LIN {X 0,Y 143.215,Z 734.624,A -85,B 0,C 180,E1 -24462.047,E2 -24462.047} C_VEL
LIN {X 0,Y 143.54,Z 734.586,A -85,B 0,C 180,E1 -24468.706,E2 -24468.706} C_VEL
LIN {X 0,Y 143.596,Z 734.591,A -85,B 0,C 180,E1 -24471.557,E2 -24471.557} C_VEL
LIN {X 0,Y 144.126,Z 734.536,A -85,B 0,C 180,E1 -24480,E2 -24480} C_VEL
LIN {X 0,Y 143.584,Z 734.584,A -85,B 0,C 180,E1 -24488.444,E2 -24488.444} C_VEL
LIN {X 0,Y 143.385,Z 734.625,A -85,B 0,C 180,E1 -24492.741,E2 -24492.741} C_VEL
LIN {X 0,Y 143.397,Z 734.844,A -85,B 0,C 180,E1 -24493.461,E2 -24493.461} C_VEL
LIN {X 0,Y 144.593,Z 738.379,A -85,B 0,C 180,E1 -24498.325,E2 -24498.325} C_VEL
LIN {X 0,Y 149.594,Z 746.195,A -85,B 0,C 180,E1 -24504.088,E2 -24504.088} C_VEL
LIN {X 0,Y 150.898,Z 748.17,A -85,B 0,C 180,E1 -24505.335,E2 -24505.335} C_VEL
LIN {X 0,Y 155.689,Z 755.868,A -85,B 0,C 180,E1 -24509.397,E2 -24509.397} C_VEL
LIN {X 0,Y 159.728,Z 762.939,A -85,B 0,C 180,E1 -24512.355,E2 -24512.355} C_VEL
LIN {X 0,Y 163.362,Z 769.766,A -85,B 0,C 180,E1 -24514.752,E2 -24514.752} C_VEL
LIN {X 0,Y 166.388,Z 775.905,A -85,B 0,C 180,E1 -24516.604,E2 -24516.604} C_VEL
LIN {X 0,Y 170.599,Z 785.165,A -85,B 0,C 180,E1 -24519.003,E2 -24519.003} C_VEL
LIN {X 0,Y 175.203,Z 796.764,A -85,B 0,C 180,E1 -24521.461,E2 -24521.461} C_VEL
LIN {X 0,Y 175.895,Z 798.887,A -85,B 0,C 180,E1 -24521.832,E2 -24521.832} C_VEL
LIN {X 0,Y 177.097,Z 822.748,A -85,B 0,C 180,E1 -24523.616,E2 -24523.616} C_VEL
LIN {X 0,Y 177.866,Z 846.501,A -85,B 0,C 180,E1 -24525.184,E2 -24525.184} C_VEL
LIN {X 0,Y 176.539,Z 862.826,A -85,B 0,C 180,E1 -24525.881,E2 -24525.881} C_VEL
LIN {X 0,Y 174.42,Z 875.839,A -85,B 0,C 180,E1 -24526.79,E2 -24526.79} C_VEL
LIN {X 0,Y 171.762,Z 887.436,A -85,B 0,C 180,E1 -24527.956,E2 -24527.956} C_VEL
LIN {X 0,Y 168.154,Z 899.75,A -85,B 0,C 180,E1 -24529.647,E2 -24529.647} C_VEL
LIN {X 0,Y 164.16,Z 910.742,A -85,B 0,C 180,E1 -24531.651,E2 -24531.651} C_VEL
LIN {X 0,Y 160.406,Z 919.713,A -85,B 0,C 180,E1 -24533.761,E2 -24533.761} C_VEL
LIN {X 0,Y 156.192,Z 928.978,A -85,B 0,C 180,E1 -24536.574,E2 -24536.574} C_VEL
LIN {X 0,Y 151.739,Z 938.048,A -85,B 0,C 180,E1 -24540.161,E2 -24540.161} C_VEL
LIN {X 0,Y 147.966,Z 945.838,A -85,B 0,C 180,E1 -24544.259,E2 -24544.259} C_VEL
LIN {X 0,Y 144.95,Z 952.191,A -85,B 0,C 180,E1 -24548.697,E2 -24548.697} C_VEL
LIN {X 0,Y 143.145,Z 956.745,A -85,B 0,C 180,E1 -24552.888,E2 -24552.888} C_VEL
LIN {X 0,Y 142.563,Z 958.65,A -85,B 0,C 180,E1 -24555.055,E2 -24555.055} C_VEL
LIN {X 0,Y 141.552,Z 960.306,A -85,B 0,C 180,E1 -24557.308,E2 -24557.308} C_VEL
LIN {X 0,Y 138.628,Z 962.218,A -85,B 0,C 180,E1 -24561.1,E2 -24561.1} C_VEL
LIN {X 0,Y 136.461,Z 963.168,A -85,B 0,C 180,E1 -24564.281,E2 -24564.281} C_VEL
LIN {X 0,Y 135.714,Z 963.596,A -85,B 0,C 180,E1 -24566.766,E2 -24566.766} C_VEL
LIN {X 0,Y 135.734,Z 963.691,A -85,B 0,C 180,E1 -24567.604,E2 -24567.604} C_VEL
LIN {X 0,Y 136.146,Z 963.933,A -85,B 0,C 180,E1 -24570.02,E2 -24570.02} C_VEL
LIN {X 0,Y 135.66,Z 963.612,A -85,B 0,C 180,E1 -24572.989,E2 -24572.989} C_VEL
LIN {X 0,Y 135.089,Z 961.834,A -85,B 0,C 180,E1 -24578.706,E2 -24578.706} C_VEL
LIN {X 0,Y 135.494,Z 959.18,A -85,B 0,C 180,E1 -24583.517,E2 -24583.517} C_VEL
LIN {X 0,Y 136.879,Z 955.695,A -85,B 0,C 180,E1 -24587.962,E2 -24587.962} C_VEL
LIN {X 0,Y 139.288,Z 951.174,A -85,B 0,C 180,E1 -24592.255,E2 -24592.255} C_VEL
LIN {X 0,Y 140.522,Z 949.425,A -85,B 0,C 180,E1 -24593.8,E2 -24593.8} C_VEL
LIN {X 0,Y 144.564,Z 949.723,A -85,B 0,C 180,E1 -24599.107,E2 -24599.107} C_VEL
LIN {X 0,Y 150.41,Z 949.085,A -85,B 0,C 180,E1 -24604.123,E2 -24604.123} C_VEL
LIN {X 0,Y 157.797,Z 947.43,A -85,B 0,C 180,E1 -24608.593,E2 -24608.593} C_VEL
LIN {X 0,Y 166.537,Z 944.767,A -85,B 0,C 180,E1 -24612.489,E2 -24612.489} C_VEL
LIN {X 0,Y 176.498,Z 941.078,A -85,B 0,C 180,E1 -24615.804,E2 -24615.804} C_VEL
LIN {X 0,Y 187.445,Z 936.242,A -85,B 0,C 180,E1 -24618.596,E2 -24618.596} C_VEL
LIN {X 0,Y 189.259,Z 935.33,A -85,B 0,C 180,E1 -24619,E2 -24619} C_VEL
LIN {X 0,Y 190.283,Z 934.518,A -85,B 0,C 180,E1 -24619.751,E2 -24619.751} C_VEL
LIN {X 0,Y 182.622,Z 935.878,A -85,B 0,C 180,E1 -24621.994,E2 -24621.994} C_VEL
LIN {X 0,Y 177.697,Z 936.442,A -85,B 0,C 180,E1 -24623.612,E2 -24623.612} C_VEL
LIN {X 0,Y 168.414,Z 936.343,A -85,B 0,C 180,E1 -24627.146,E2 -24627.146} C_VEL
LIN {X 0,Y 160.138,Z 934.838,A -85,B 0,C 180,E1 -24631.134,E2 -24631.134} C_VEL
LIN {X 0,Y 156.316,Z 933.555,A -85,B 0,C 180,E1 -24633.282,E2 -24633.282} C_VEL
LIN {X 0,Y 149.601,Z 929.833,A -85,B 0,C 180,E1 -24637.925,E2 -24637.925} C_VEL
LIN {X 0,Y 145.372,Z 926.105,A -85,B 0,C 180,E1 -24641.685,E2 -24641.685} C_VEL
LIN {X 0,Y 142.096,Z 921.514,A -85,B 0,C 180,E1 -24645.682,E2 -24645.682} C_VEL
LIN {X 0,Y 139.213,Z 914.828,A -85,B 0,C 180,E1 -24650.557,E2 -24650.557} C_VEL
LIN {X 0,Y 137.471,Z 907.937,A -85,B 0,C 180,E1 -24654.867,E2 -24654.867} C_VEL
LIN {X 0,Y 136.486,Z 899.695,A -85,B 0,C 180,E1 -24659.263,E2 -24659.263} C_VEL
LIN {X 0,Y 136.223,Z 891.671,A -85,B 0,C 180,E1 -24662.957,E2 -24662.957} C_VEL
LIN {X 0,Y 136.591,Z 882.287,A -85,B 0,C 180,E1 -24666.648,E2 -24666.648} C_VEL
LIN {X 0,Y 137.066,Z 872.251,A -85,B 0,C 180,E1 -24669.965,E2 -24669.965} C_VEL
LIN {X 0,Y 137.976,Z 859.138,A -85,B 0,C 180,E1 -24673.564,E2 -24673.564} C_VEL
LIN {X 0,Y 138.76,Z 846.996,A -85,B 0,C 180,E1 -24676.173,E2 -24676.173} C_VEL
LIN {X 0,Y 139.713,Z 834.461,A -85,B 0,C 180,E1 -24678.324,E2 -24678.324} C_VEL
LIN {X 0,Y 140.393,Z 821.589,A -85,B 0,C 180,E1 -24680.035,E2 -24680.035} C_VEL
LIN {X 0,Y 141.461,Z 793.316,A -85,B 0,C 180,E1 -24682.839,E2 -24682.839} C_VEL
LIN {X 0,Y 141.712,Z 783.104,A -85,B 0,C 180,E1 -24683.831,E2 -24683.831} C_VEL
LIN {X 0,Y 141.993,Z 785.657,A -85,B 0,C 180,E1 -24684.419,E2 -24684.419} C_VEL
LIN {X 0,Y 142.462,Z 785.901,A -85,B 0,C 180,E1 -24684.881,E2 -24684.881} C_VEL
LIN {X 0,Y 143.783,Z 783.644,A -85,B 0,C 180,E1 -24685.783,E2 -24685.783} C_VEL
LIN {X 0,Y 145.983,Z 777.23,A -85,B 0,C 180,E1 -24686.894,E2 -24686.894} C_VEL
LIN {X 0,Y 149.817,Z 763.086,A -85,B 0,C 180,E1 -24688.358,E2 -24688.358} C_VEL
LIN {X 0,Y 151.85,Z 761.187,A -85,B 0,C 180,E1 -24689.624,E2 -24689.624} C_VEL
LIN {X 0,Y 153.83,Z 757.884,A -85,B 0,C 180,E1 -24690.644,E2 -24690.644} C_VEL
LIN {X 0,Y 153.971,Z 757.58,A -85,B 0,C 180,E1 -24690.708,E2 -24690.708} C_VEL
LIN {X 0,Y 157.697,Z 762.748,A -85,B 0,C 180,E1 -24693.436,E2 -24693.436} C_VEL
LIN {X 0,Y 162.667,Z 770.012,A -85,B 0,C 180,E1 -24696.64,E2 -24696.64} C_VEL
LIN {X 0,Y 168.766,Z 780.01,A -85,B 0,C 180,E1 -24700.103,E2 -24700.103} C_VEL
LIN {X 0,Y 174.092,Z 790.072,A -85,B 0,C 180,E1 -24702.828,E2 -24702.828} C_VEL
LIN {X 0,Y 176.12,Z 794.353,A -85,B 0,C 180,E1 -24703.813,E2 -24703.813} C_VEL
LIN {X 0,Y 174.707,Z 823.428,A -85,B 0,C 180,E1 -24705.124,E2 -24705.124} C_VEL
LIN {X 0,Y 173.298,Z 836.373,A -85,B 0,C 180,E1 -24706.097,E2 -24706.097} C_VEL
LIN {X 0,Y 171.192,Z 848.235,A -85,B 0,C 180,E1 -24707.345,E2 -24707.345} C_VEL
LIN {X 0,Y 168.406,Z 859.637,A -85,B 0,C 180,E1 -24708.943,E2 -24708.943} C_VEL
LIN {X 0,Y 164.85,Z 870.933,A -85,B 0,C 180,E1 -24711.019,E2 -24711.019} C_VEL
LIN {X 0,Y 161.046,Z 881.241,A -85,B 0,C 180,E1 -24713.499,E2 -24713.499} C_VEL
LIN {X 0,Y 157.524,Z 889.637,A -85,B 0,C 180,E1 -24716.086,E2 -24716.086} C_VEL
LIN {X 0,Y 153.752,Z 897.386,A -85,B 0,C 180,E1 -24719.036,E2 -24719.036} C_VEL
LIN {X 0,Y 149.632,Z 905.052,A -85,B 0,C 180,E1 -24722.803,E2 -24722.803} C_VEL
LIN {X 0,Y 146.452,Z 910.677,A -85,B 0,C 180,E1 -24726.412,E2 -24726.412} C_VEL
LIN {X 0,Y 143.01,Z 916.427,A -85,B 0,C 180,E1 -24731.353,E2 -24731.353} C_VEL
LIN {X 0,Y 140.439,Z 919.981,A -85,B 0,C 180,E1 -24735.491,E2 -24735.491} C_VEL
LIN {X 0,Y 139.187,Z 921.802,A -85,B 0,C 180,E1 -24738.329,E2 -24738.329} C_VEL
LIN {X 0,Y 137.812,Z 924.102,A -85,B 0,C 180,E1 -24744.127,E2 -24744.127} C_VEL
LIN {X 0,Y 137.196,Z 924.935,A -85,B 0,C 180,E1 -24749.981,E2 -24749.981} C_VEL
LIN {X 0,Y 137.801,Z 924.164,A -85,B 0,C 180,E1 -24755.835,E2 -24755.835} C_VEL
LIN {X 0,Y 139.154,Z 921.929,A -85,B 0,C 180,E1 -24761.635,E2 -24761.635} C_VEL
LIN {X 0,Y 141.179,Z 919.101,A -85,B 0,C 180,E1 -24765.869,E2 -24765.869} C_VEL
LIN {X 0,Y 143.796,Z 915.268,A -85,B 0,C 180,E1 -24769.985,E2 -24769.985} C_VEL
LIN {X 0,Y 147.043,Z 909.785,A -85,B 0,C 180,E1 -24774.415,E2 -24774.415} C_VEL
LIN {X 0,Y 150.924,Z 902.963,A -85,B 0,C 180,E1 -24778.487,E2 -24778.487} C_VEL
LIN {X 0,Y 155.166,Z 894.923,A -85,B 0,C 180,E1 -24782.131,E2 -24782.131} C_VEL
LIN {X 0,Y 158.973,Z 886.69,A -85,B 0,C 180,E1 -24785.056,E2 -24785.056} C_VEL
LIN {X 0,Y 163.049,Z 876.498,A -85,B 0,C 180,E1 -24787.872,E2 -24787.872} C_VEL
LIN {X 0,Y 166.719,Z 866.009,A -85,B 0,C 180,E1 -24790.084,E2 -24790.084} C_VEL
LIN {X 0,Y 169.93,Z 854.712,A -85,B 0,C 180,E1 -24791.932,E2 -24791.932} C_VEL
LIN {X 0,Y 172.59,Z 842.714,A -85,B 0,C 180,E1 -24793.38,E2 -24793.38} C_VEL
LIN {X 0,Y 174.299,Z 829.63,A -85,B 0,C 180,E1 -24794.611,E2 -24794.611} C_VEL
LIN {X 0,Y 175.304,Z 816.492,A -85,B 0,C 180,E1 -24795.384,E2 -24795.384} C_VEL
LIN {X 0,Y 176.319,Z 794.58,A -85,B 0,C 180,E1 -24796.312,E2 -24796.312} C_VEL
LIN {X 0,Y 171.395,Z 784.61,A -85,B 0,C 180,E1 -24798.756,E2 -24798.756} C_VEL
LIN {X 0,Y 165.956,Z 775.095,A -85,B 0,C 180,E1 -24801.687,E2 -24801.687} C_VEL
LIN {X 0,Y 161.641,Z 768.383,A -85,B 0,C 180,E1 -24804.25,E2 -24804.25} C_VEL
LIN {X 0,Y 156.965,Z 761.488,A -85,B 0,C 180,E1 -24807.374,E2 -24807.374} C_VEL
LIN {X 0,Y 154.139,Z 757.622,A -85,B 0,C 180,E1 -24809.478,E2 -24809.478} C_VEL
LIN {X 0,Y 151.045,Z 753.831,A -85,B 0,C 180,E1 -24812.006,E2 -24812.006} C_VEL
LIN {X 0,Y 150.012,Z 752.328,A -85,B 0,C 180,E1 -24812.951,E2 -24812.951} C_VEL
LIN {X 0,Y 147.477,Z 749.672,A -85,B 0,C 180,E1 -24815.356,E2 -24815.356} C_VEL
LIN {X 0,Y 146.05,Z 747.186,A -85,B 0,C 180,E1 -24816.984,E2 -24816.984} C_VEL
LIN {X 0,Y 143.499,Z 745.206,A -85,B 0,C 180,E1 -24819.95,E2 -24819.95} C_VEL
LIN {X 0,Y 141.928,Z 742.484,A -85,B 0,C 180,E1 -24822.344,E2 -24822.344} C_VEL
LIN {X 0,Y 141.547,Z 741.518,A -85,B 0,C 180,E1 -24823.04,E2 -24823.04} C_VEL
LIN {X 0,Y 139.001,Z 740.155,A -85,B 0,C 180,E1 -24827.591,E2 -24827.591} C_VEL
LIN {X 0,Y 136.829,Z 736.174,A -85,B 0,C 180,E1 -24836.871,E2 -24836.871} C_VEL
LIN {X 0,Y 136.88,Z 735.432,A -85,B 0,C 180,E1 -24838.529,E2 -24838.529} C_VEL
LIN {X 0,Y 136.939,Z 735.42,A -85,B 0,C 180,E1 -24840.919,E2 -24840.919} C_VEL
LIN {X 0,Y 137.547,Z 738.415,A -85,B 0,C 180,E1 -24846.233,E2 -24846.233} C_VEL
LIN {X 0,Y 140.29,Z 741.186,A -85,B 0,C 180,E1 -24853.028,E2 -24853.028} C_VEL
LIN {X 0,Y 142.855,Z 744.781,A -85,B 0,C 180,E1 -24857.26,E2 -24857.26} C_VEL
LIN {X 0,Y 148.531,Z 754.019,A -85,B 0,C 180,E1 -24864.086,E2 -24864.086} C_VEL
LIN {X 0,Y 153.085,Z 761.749,A -85,B 0,C 180,E1 -24868.249,E2 -24868.249} C_VEL
LIN {X 0,Y 156.942,Z 768.865,A -85,B 0,C 180,E1 -24871.277,E2 -24871.277} C_VEL
LIN {X 0,Y 160.558,Z 775.925,A -85,B 0,C 180,E1 -24873.813,E2 -24873.813} C_VEL
LIN {X 0,Y 164.724,Z 784.987,A -85,B 0,C 180,E1 -24876.488,E2 -24876.488} C_VEL
LIN {X 0,Y 169.168,Z 795.925,A -85,B 0,C 180,E1 -24879.121,E2 -24879.121} C_VEL
LIN {X 0,Y 171.175,Z 801.56,A -85,B 0,C 180,E1 -24880.265,E2 -24880.265} C_VEL
LIN {X 0,Y 172.232,Z 825.486,A -85,B 0,C 180,E1 -24882.114,E2 -24882.114} C_VEL
LIN {X 0,Y 172.771,Z 847.209,A -85,B 0,C 180,E1 -24883.58,E2 -24883.58} C_VEL
LIN {X 0,Y 171.528,Z 861.709,A -85,B 0,C 180,E1 -24884.224,E2 -24884.224} C_VEL
LIN {X 0,Y 169.333,Z 874.838,A -85,B 0,C 180,E1 -24885.151,E2 -24885.151} C_VEL
LIN {X 0,Y 166.568,Z 886.431,A -85,B 0,C 180,E1 -24886.324,E2 -24886.324} C_VEL
LIN {X 0,Y 162.78,Z 898.737,A -85,B 0,C 180,E1 -24888.02,E2 -24888.02} C_VEL
LIN {X 0,Y 158.656,Z 909.733,A -85,B 0,C 180,E1 -24890.061,E2 -24890.061} C_VEL
LIN {X 0,Y 154.736,Z 918.703,A -85,B 0,C 180,E1 -24892.206,E2 -24892.206} C_VEL
LIN {X 0,Y 150.287,Z 927.962,A -85,B 0,C 180,E1 -24895.075,E2 -24895.075} C_VEL
LIN {X 0,Y 145.582,Z 937.03,A -85,B 0,C 180,E1 -24898.761,E2 -24898.761} C_VEL
LIN {X 0,Y 141.77,Z 944.4,A -85,B 0,C 180,E1 -24902.73,E2 -24902.73} C_VEL
LIN {X 0,Y 138.291,Z 951.169,A -85,B 0,C 180,E1 -24907.617,E2 -24907.617} C_VEL
LIN {X 0,Y 136.302,Z 955.723,A -85,B 0,C 180,E1 -24912,E2 -24912} C_VEL
LIN {X 0,Y 135.225,Z 959.226,A -85,B 0,C 180,E1 -24916.496,E2 -24916.496} C_VEL
LIN {X 0,Y 135.034,Z 961.93,A -85,B 0,C 180,E1 -24921.447,E2 -24921.447} C_VEL
LIN {X 0,Y 135.261,Z 962.903,A -85,B 0,C 180,E1 -24924.055,E2 -24924.055} C_VEL
LIN {X 0,Y 135.734,Z 963.691,A -85,B 0,C 180,E1 -24927.604,E2 -24927.604} C_VEL
LIN {X 0,Y 135.525,Z 963.812,A -85,B 0,C 180,E1 -24929.253,E2 -24929.253} C_VEL
LIN {X 0,Y 134.689,Z 963.68,A -85,B 0,C 180,E1 -24930.879,E2 -24930.879} C_VEL
LIN {X 0,Y 132.014,Z 962.911,A -85,B 0,C 180,E1 -24934.087,E2 -24934.087} C_VEL
LIN {X 0,Y 129.242,Z 961.659,A -85,B 0,C 180,E1 -24937.416,E2 -24937.416} C_VEL
LIN {X 0,Y 128.079,Z 960.262,A -85,B 0,C 180,E1 -24940.469,E2 -24940.469} C_VEL
LIN {X 0,Y 128.082,Z 959.996,A -85,B 0,C 180,E1 -24940.912,E2 -24940.912} C_VEL
LIN {X 0,Y 128.957,Z 957.11,A -85,B 0,C 180,E1 -24945.833,E2 -24945.833} C_VEL
LIN {X 0,Y 130.85,Z 953.292,A -85,B 0,C 180,E1 -24950.454,E2 -24950.454} C_VEL
LIN {X 0,Y 134.708,Z 947.373,A -85,B 0,C 180,E1 -24955.722,E2 -24955.722} C_VEL
LIN {X 0,Y 138.574,Z 947.822,A -85,B 0,C 180,E1 -24960.495,E2 -24960.495} C_VEL
LIN {X 0,Y 144.692,Z 947.513,A -85,B 0,C 180,E1 -24965.672,E2 -24965.672} C_VEL
LIN {X 0,Y 152.37,Z 946.329,A -85,B 0,C 180,E1 -24970.241,E2 -24970.241} C_VEL
LIN {X 0,Y 161.391,Z 944.159,A -85,B 0,C 180,E1 -24974.185,E2 -24974.185} C_VEL
LIN {X 0,Y 171.625,Z 940.936,A -85,B 0,C 180,E1 -24977.503,E2 -24977.503} C_VEL
LIN {X 0,Y 178.622,Z 938.425,A -85,B 0,C 180,E1 -24979.312,E2 -24979.312} C_VEL
LIN {X 0,Y 179.484,Z 937.82,A -85,B 0,C 180,E1 -24979.981,E2 -24979.981} C_VEL
LIN {X 0,Y 167.27,Z 938.132,A -85,B 0,C 180,E1 -24983.969,E2 -24983.969} C_VEL
LIN {X 0,Y 158.135,Z 936.786,A -85,B 0,C 180,E1 -24987.77,E2 -24987.77} C_VEL
LIN {X 0,Y 153.993,Z 935.59,A -85,B 0,C 180,E1 -24989.866,E2 -24989.866} C_VEL
LIN {X 0,Y 146.344,Z 932.155,A -85,B 0,C 180,E1 -24994.392,E2 -24994.392} C_VEL
LIN {X 0,Y 140.044,Z 927.186,A -85,B 0,C 180,E1 -24999.434,E2 -24999.434} C_VEL
LIN {X 0,Y 136.277,Z 922.478,A -85,B 0,C 180,E1 -25003.522,E2 -25003.522} C_VEL
LIN {X 0,Y 133.052,Z 915.781,A -85,B 0,C 180,E1 -25008.575,E2 -25008.575} C_VEL
LIN {X 0,Y 131.026,Z 908.831,A -85,B 0,C 180,E1 -25013.068,E2 -25013.068} C_VEL
LIN {X 0,Y 129.889,Z 902.11,A -85,B 0,C 180,E1 -25016.898,E2 -25016.898} C_VEL
LIN {X 0,Y 129.377,Z 894.283,A -85,B 0,C 180,E1 -25020.778,E2 -25020.778} C_VEL
LIN {X 0,Y 129.42,Z 885.191,A -85,B 0,C 180,E1 -25024.672,E2 -25024.672} C_VEL
LIN {X 0,Y 129.855,Z 876.862,A -85,B 0,C 180,E1 -25027.776,E2 -25027.776} C_VEL
LIN {X 0,Y 130.398,Z 866.955,A -85,B 0,C 180,E1 -25030.874,E2 -25030.874} C_VEL
LIN {X 0,Y 131.088,Z 856.762,A -85,B 0,C 180,E1 -25033.559,E2 -25033.559} C_VEL
LIN {X 0,Y 131.642,Z 848.197,A -85,B 0,C 180,E1 -25035.482,E2 -25035.482} C_VEL
LIN {X 0,Y 132.509,Z 836.397,A -85,B 0,C 180,E1 -25037.677,E2 -25037.677} C_VEL
LIN {X 0,Y 133.229,Z 824.283,A -85,B 0,C 180,E1 -25039.451,E2 -25039.451} C_VEL
LIN {X 0,Y 133.399,Z 819.791,A -85,B 0,C 180,E1 -25040.026,E2 -25040.026} C_VEL
LIN {X 0,Y 133.401,Z 822.286,A -85,B 0,C 180,E1 -25040.428,E2 -25040.428} C_VEL
LIN {X 0,Y 133.616,Z 822.978,A -85,B 0,C 180,E1 -25040.796,E2 -25040.796} C_VEL
LIN {X 0,Y 134.191,Z 822.56,A -85,B 0,C 180,E1 -25041.406,E2 -25041.406} C_VEL
LIN {X 0,Y 135.462,Z 819.648,A -85,B 0,C 180,E1 -25042.396,E2 -25042.396} C_VEL
LIN {X 0,Y 137.846,Z 811.695,A -85,B 0,C 180,E1 -25043.772,E2 -25043.772} C_VEL
LIN {X 0,Y 141.268,Z 798.31,A -85,B 0,C 180,E1 -25045.31,E2 -25045.31} C_VEL
LIN {X 0,Y 142.632,Z 792.59,A -85,B 0,C 180,E1 -25045.834,E2 -25045.834} C_VEL
LIN {X 0,Y 144.333,Z 790.543,A -85,B 0,C 180,E1 -25047.03,E2 -25047.03} C_VEL
LIN {X 0,Y 146.121,Z 787.039,A -85,B 0,C 180,E1 -25048.064,E2 -25048.064} C_VEL
LIN {X 0,Y 148.597,Z 780.127,A -85,B 0,C 180,E1 -25049.192,E2 -25049.192} C_VEL
LIN {X 0,Y 152.084,Z 768.248,A -85,B 0,C 180,E1 -25050.456,E2 -25050.456} C_VEL
LIN {X 0,Y 153.197,Z 766.995,A -85,B 0,C 180,E1 -25051.071,E2 -25051.071} C_VEL
LIN {X 0,Y 154.267,Z 767.394,A -85,B 0,C 180,E1 -25051.787,E2 -25051.787} C_VEL
LIN {X 0,Y 159.68,Z 775.763,A -85,B 0,C 180,E1 -25055.565,E2 -25055.565} C_VEL
LIN {X 0,Y 165.269,Z 785.185,A -85,B 0,C 180,E1 -25058.945,E2 -25058.945} C_VEL
LIN {X 0,Y 170.645,Z 795.676,A -85,B 0,C 180,E1 -25061.871,E2 -25061.871} C_VEL
LIN {X 0,Y 171.251,Z 796.983,A -85,B 0,C 180,E1 -25062.186,E2 -25062.186} C_VEL
LIN {X 0,Y 169.777,Z 824.796,A -85,B 0,C 180,E1 -25063.476,E2 -25063.476} C_VEL
LIN {X 0,Y 168.208,Z 838.025,A -85,B 0,C 180,E1 -25064.495,E2 -25064.495} C_VEL
LIN {X 0,Y 165.809,Z 850.431,A -85,B 0,C 180,E1 -25065.839,E2 -25065.839} C_VEL
LIN {X 0,Y 162.821,Z 861.789,A -85,B 0,C 180,E1 -25067.516,E2 -25067.516} C_VEL
LIN {X 0,Y 158.984,Z 873.211,A -85,B 0,C 180,E1 -25069.702,E2 -25069.702} C_VEL
LIN {X 0,Y 155.02,Z 883.291,A -85,B 0,C 180,E1 -25072.244,E2 -25072.244} C_VEL
LIN {X 0,Y 150.93,Z 892.311,A -85,B 0,C 180,E1 -25075.202,E2 -25075.202} C_VEL
LIN {X 0,Y 146.263,Z 901.085,A -85,B 0,C 180,E1 -25078.881,E2 -25078.881} C_VEL
LIN {X 0,Y 141.775,Z 908.743,A -85,B 0,C 180,E1 -25083.163,E2 -25083.163} C_VEL
LIN {X 0,Y 138.281,Z 914.499,A -85,B 0,C 180,E1 -25087.574,E2 -25087.574} C_VEL
LIN {X 0,Y 136.369,Z 917.431,A -85,B 0,C 180,E1 -25090.409,E2 -25090.409} C_VEL
LIN {X 0,Y 133.647,Z 920.984,A -85,B 0,C 180,E1 -25094.736,E2 -25094.736} C_VEL
LIN {X 0,Y 132.312,Z 922.805,A -85,B 0,C 180,E1 -25097.713,E2 -25097.713} C_VEL
LIN {X 0,Y 130.823,Z 925.105,A -85,B 0,C 180,E1 -25103.812,E2 -25103.812} C_VEL
LIN {X 0,Y 130.168,Z 925.938,A -85,B 0,C 180,E1 -25109.979,E2 -25109.979} C_VEL
LIN {X 0,Y 130.811,Z 925.166,A -85,B 0,C 180,E1 -25116.148,E2 -25116.148} C_VEL
LIN {X 0,Y 132.277,Z 922.931,A -85,B 0,C 180,E1 -25122.249,E2 -25122.249} C_VEL
LIN {X 0,Y 134.432,Z 920.103,A -85,B 0,C 180,E1 -25126.688,E2 -25126.688} C_VEL
LIN {X 0,Y 137.212,Z 916.27,A -85,B 0,C 180,E1 -25130.988,E2 -25130.988} C_VEL
LIN {X 0,Y 140.674,Z 910.786,A -85,B 0,C 180,E1 -25135.598,E2 -25135.598} C_VEL
LIN {X 0,Y 144.785,Z 903.963,A -85,B 0,C 180,E1 -25139.814,E2 -25139.814} C_VEL
LIN {X 0,Y 149.262,Z 895.924,A -85,B 0,C 180,E1 -25143.566,E2 -25143.566} C_VEL
LIN {X 0,Y 153.273,Z 887.69,A -85,B 0,C 180,E1 -25146.565,E2 -25146.565} C_VEL
LIN {X 0,Y 157.56,Z 877.497,A -85,B 0,C 180,E1 -25149.441,E2 -25149.441} C_VEL
LIN {X 0,Y 161.405,Z 867.007,A -85,B 0,C 180,E1 -25151.69,E2 -25151.69} C_VEL
LIN {X 0,Y 164.916,Z 855.171,A -85,B 0,C 180,E1 -25153.642,E2 -25153.642} C_VEL
LIN {X 0,Y 167.703,Z 842.562,A -85,B 0,C 180,E1 -25155.171,E2 -25155.171} C_VEL
LIN {X 0,Y 169.481,Z 829.62,A -85,B 0,C 180,E1 -25156.36,E2 -25156.36} C_VEL
LIN {X 0,Y 170.461,Z 816.623,A -85,B 0,C 180,E1 -25157.111,E2 -25157.111} C_VEL
LIN {X 0,Y 171.369,Z 797.105,A -85,B 0,C 180,E1 -25157.979,E2 -25157.979} C_VEL
LIN {X 0,Y 166.368,Z 787.041,A -85,B 0,C 180,E1 -25160.679,E2 -25160.679} C_VEL
LIN {X 0,Y 161.086,Z 777.773,A -85,B 0,C 180,E1 -25163.818,E2 -25163.818} C_VEL
LIN {X 0,Y 156.342,Z 770.49,A -85,B 0,C 180,E1 -25166.975,E2 -25166.975} C_VEL
LIN {X 0,Y 153.448,Z 766.362,A -85,B 0,C 180,E1 -25169.123,E2 -25169.123} C_VEL
LIN {X 0,Y 151.179,Z 763.125,A -85,B 0,C 180,E1 -25170.973,E2 -25170.973} C_VEL
LIN {X 0,Y 148.425,Z 759.301,A -85,B 0,C 180,E1 -25173.455,E2 -25173.455} C_VEL
LIN {X 0,Y 145.354,Z 755.708,A -85,B 0,C 180,E1 -25176.567,E2 -25176.567} C_VEL
LIN {X 0,Y 144.34,Z 753.876,A -85,B 0,C 180,E1 -25177.807,E2 -25177.807} C_VEL
LIN {X 0,Y 141.781,Z 751.609,A -85,B 0,C 180,E1 -25181.016,E2 -25181.016} C_VEL
LIN {X 0,Y 140.032,Z 748.394,A -85,B 0,C 180,E1 -25183.976,E2 -25183.976} C_VEL
LIN {X 0,Y 137.553,Z 746.665,A -85,B 0,C 180,E1 -25188.976,E2 -25188.976} C_VEL
LIN {X 0,Y 135.942,Z 742.879,A -85,B 0,C 180,E1 -25197.778,E2 -25197.778} C_VEL
LIN {X 0,Y 135.964,Z 742.479,A -85,B 0,C 180,E1 -25198.519,E2 -25198.519} C_VEL
LIN {X 0,Y 136.01,Z 742.681,A -85,B 0,C 180,E1 -25200.925,E2 -25200.925} C_VEL
LIN {X 0,Y 136.586,Z 745.399,A -85,B 0,C 180,E1 -25205.907,E2 -25205.907} C_VEL
LIN {X 0,Y 139.05,Z 748.068,A -85,B 0,C 180,E1 -25212.404,E2 -25212.404} C_VEL
LIN {X 0,Y 141.321,Z 751.539,A -85,B 0,C 180,E1 -25216.43,E2 -25216.43} C_VEL
LIN {X 0,Y 146.31,Z 760.01,A -85,B 0,C 180,E1 -25222.879,E2 -25222.879} C_VEL
LIN {X 0,Y 150.554,Z 767.686,A -85,B 0,C 180,E1 -25227.074,E2 -25227.074} C_VEL
LIN {X 0,Y 153.943,Z 774.202,A -85,B 0,C 180,E1 -25229.94,E2 -25229.94} C_VEL
LIN {X 0,Y 157.337,Z 781.098,A -85,B 0,C 180,E1 -25232.509,E2 -25232.509} C_VEL
LIN {X 0,Y 161.577,Z 790.876,A -85,B 0,C 180,E1 -25235.44,E2 -25235.44} C_VEL
LIN {X 0,Y 165.192,Z 800.277,A -85,B 0,C 180,E1 -25237.752,E2 -25237.752} C_VEL
LIN {X 0,Y 166.626,Z 804.842,A -85,B 0,C 180,E1 -25238.665,E2 -25238.665} C_VEL
LIN {X 0,Y 167.449,Z 827.771,A -85,B 0,C 180,E1 -25240.48,E2 -25240.48} C_VEL
LIN {X 0,Y 167.822,Z 847.922,A -85,B 0,C 180,E1 -25241.881,E2 -25241.881} C_VEL
LIN {X 0,Y 166.497,Z 861.823,A -85,B 0,C 180,E1 -25242.534,E2 -25242.534} C_VEL
LIN {X 0,Y 164.081,Z 875.139,A -85,B 0,C 180,E1 -25243.519,E2 -25243.519} C_VEL
LIN {X 0,Y 160.916,Z 887.42,A -85,B 0,C 180,E1 -25244.816,E2 -25244.816} C_VEL
LIN {X 0,Y 157.012,Z 899.252,A -85,B 0,C 180,E1 -25246.539,E2 -25246.539} C_VEL
LIN {X 0,Y 152.746,Z 909.906,A -85,B 0,C 180,E1 -25248.619,E2 -25248.619} C_VEL
LIN {X 0,Y 148.191,Z 919.665,A -85,B 0,C 180,E1 -25251.095,E2 -25251.095} C_VEL
LIN {X 0,Y 143.621,Z 928.603,A -85,B 0,C 180,E1 -25254.066,E2 -25254.066} C_VEL
LIN {X 0,Y 138.778,Z 937.358,A -85,B 0,C 180,E1 -25257.902,E2 -25257.902} C_VEL
LIN {X 0,Y 134.856,Z 944.436,A -85,B 0,C 180,E1 -25262.053,E2 -25262.053} C_VEL
LIN {X 0,Y 131.695,Z 950.148,A -85,B 0,C 180,E1 -25266.43,E2 -25266.43} C_VEL
LIN {X 0,Y 129.499,Z 954.7,A -85,B 0,C 180,E1 -25271.02,E2 -25271.02} C_VEL
LIN {X 0,Y 128.266,Z 958.204,A -85,B 0,C 180,E1 -25275.748,E2 -25275.748} C_VEL
LIN {X 0,Y 127.968,Z 961.053,A -85,B 0,C 180,E1 -25281.327,E2 -25281.327} C_VEL
LIN {X 0,Y 128.595,Z 962.625,A -85,B 0,C 180,E1 -25286.888,E2 -25286.888} C_VEL
LIN {X 0,Y 129.082,Z 962.925,A -85,B 0,C 180,E1 -25290.021,E2 -25290.021} C_VEL
LIN {X 0,Y 128.584,Z 962.601,A -85,B 0,C 180,E1 -25293.154,E2 -25293.154} C_VEL
LIN {X 0,Y 128.032,Z 960.948,A -85,B 0,C 180,E1 -25298.859,E2 -25298.859} C_VEL
LIN {X 0,Y 128.082,Z 959.996,A -85,B 0,C 180,E1 -25300.912,E2 -25300.912} C_VEL
LIN {X 0,Y 127.722,Z 958.597,A -85,B 0,C 180,E1 -25303.479,E2 -25303.479} C_VEL
LIN {X 0,Y 125.964,Z 955.605,A -85,B 0,C 180,E1 -25307.689,E2 -25307.689} C_VEL
LIN {X 0,Y 125.049,Z 952.018,A -85,B 0,C 180,E1 -25311.878,E2 -25311.878} C_VEL
LIN {X 0,Y 125.987,Z 949.585,A -85,B 0,C 180,E1 -25314.289,E2 -25314.289} C_VEL
LIN {X 0,Y 129.316,Z 945.102,A -85,B 0,C 180,E1 -25317.974,E2 -25317.974} C_VEL
LIN {X 0,Y 135.709,Z 945.881,A -85,B 0,C 180,E1 -25324.748,E2 -25324.748} C_VEL
LIN {X 0,Y 142.95,Z 945.506,A -85,B 0,C 180,E1 -25329.748,E2 -25329.748} C_VEL
LIN {X 0,Y 151.572,Z 944.277,A -85,B 0,C 180,E1 -25334.089,E2 -25334.089} C_VEL
LIN {X 0,Y 161.552,Z 942.131,A -85,B 0,C 180,E1 -25337.713,E2 -25337.713} C_VEL
LIN {X 0,Y 168.062,Z 940.336,A -85,B 0,C 180,E1 -25339.604,E2 -25339.604} C_VEL
LIN {X 0,Y 168.026,Z 939.917,A -85,B 0,C 180,E1 -25340.387,E2 -25340.387} C_VEL
LIN {X 0,Y 161.661,Z 939.494,A -85,B 0,C 180,E1 -25342.509,E2 -25342.509} C_VEL
LIN {X 0,Y 152.218,Z 937.596,A -85,B 0,C 180,E1 -25346.355,E2 -25346.355} C_VEL
LIN {X 0,Y 143.771,Z 934.325,A -85,B 0,C 180,E1 -25350.736,E2 -25350.736} C_VEL
LIN {X 0,Y 136.538,Z 929.656,A -85,B 0,C 180,E1 -25355.683,E2 -25355.683} C_VEL
LIN {X 0,Y 130.679,Z 923.393,A -85,B 0,C 180,E1 -25361.175,E2 -25361.175} C_VEL
LIN {X 0,Y 127.473,Z 917.67,A -85,B 0,C 180,E1 -25365.635,E2 -25365.635} C_VEL
LIN {X 0,Y 125.046,Z 910.925,A -85,B 0,C 180,E1 -25370.293,E2 -25370.293} C_VEL
LIN {X 0,Y 123.354,Z 902.854,A -85,B 0,C 180,E1 -25375.098,E2 -25375.098} C_VEL
LIN {X 0,Y 122.608,Z 895.048,A -85,B 0,C 180,E1 -25379.179,E2 -25379.179} C_VEL
LIN {X 0,Y 122.431,Z 887.959,A -85,B 0,C 180,E1 -25382.468,E2 -25382.468} C_VEL
LIN {X 0,Y 122.876,Z 877.627,A -85,B 0,C 180,E1 -25386.569,E2 -25386.569} C_VEL
LIN {X 0,Y 123.338,Z 867.818,A -85,B 0,C 180,E1 -25389.843,E2 -25389.843} C_VEL
LIN {X 0,Y 123.984,Z 857.77,A -85,B 0,C 180,E1 -25392.689,E2 -25392.689} C_VEL
LIN {X 0,Y 124.591,Z 848.905,A -85,B 0,C 180,E1 -25394.799,E2 -25394.799} C_VEL
LIN {X 0,Y 124.526,Z 850.104,A -85,B 0,C 180,E1 -25395.459,E2 -25395.459} C_VEL
LIN {X 0,Y 124.971,Z 850.143,A -85,B 0,C 180,E1 -25396.331,E2 -25396.331} C_VEL
LIN {X 0,Y 126.2,Z 848.449,A -85,B 0,C 180,E1 -25397.602,E2 -25397.602} C_VEL
LIN {X 0,Y 128.658,Z 843.796,A -85,B 0,C 180,E1 -25399.34,E2 -25399.34} C_VEL
LIN {X 0,Y 131.745,Z 835.961,A -85,B 0,C 180,E1 -25401.003,E2 -25401.003} C_VEL
LIN {X 0,Y 133.708,Z 829.729,A -85,B 0,C 180,E1 -25401.994,E2 -25401.994} C_VEL
LIN {X 0,Y 135.029,Z 828.246,A -85,B 0,C 180,E1 -25403.18,E2 -25403.18} C_VEL
LIN {X 0,Y 136.793,Z 824.774,A -85,B 0,C 180,E1 -25404.45,E2 -25404.45} C_VEL
LIN {X 0,Y 138.915,Z 818.716,A -85,B 0,C 180,E1 -25405.669,E2 -25405.669} C_VEL
LIN {X 0,Y 142.579,Z 805.843,A -85,B 0,C 180,E1 -25407.305,E2 -25407.305} C_VEL
LIN {X 0,Y 144.806,Z 797.334,A -85,B 0,C 180,E1 -25408.143,E2 -25408.143} C_VEL
LIN {X 0,Y 147.269,Z 793.507,A -85,B 0,C 180,E1 -25409.579,E2 -25409.579} C_VEL
LIN {X 0,Y 149.812,Z 787.701,A -85,B 0,C 180,E1 -25410.773,E2 -25410.773} C_VEL
LIN {X 0,Y 152.887,Z 778.468,A -85,B 0,C 180,E1 -25411.914,E2 -25411.914} C_VEL
LIN {X 0,Y 153.562,Z 776.326,A -85,B 0,C 180,E1 -25412.143,E2 -25412.143} C_VEL
LIN {X 0,Y 158.592,Z 784.519,A -85,B 0,C 180,E1 -25415.678,E2 -25415.678} C_VEL
LIN {X 0,Y 163.748,Z 794.047,A -85,B 0,C 180,E1 -25418.881,E2 -25418.881} C_VEL
LIN {X 0,Y 166.502,Z 799.825,A -85,B 0,C 180,E1 -25420.47,E2 -25420.47} C_VEL
LIN {X 0,Y 165.065,Z 825.382,A -85,B 0,C 180,E1 -25421.679,E2 -25421.679} C_VEL
LIN {X 0,Y 163.446,Z 838.52,A -85,B 0,C 180,E1 -25422.692,E2 -25422.692} C_VEL
LIN {X 0,Y 161.135,Z 850.256,A -85,B 0,C 180,E1 -25423.956,E2 -25423.956} C_VEL
LIN {X 0,Y 157.961,Z 862.006,A -85,B 0,C 180,E1 -25425.654,E2 -25425.654} C_VEL
LIN {X 0,Y 154.178,Z 872.947,A -85,B 0,C 180,E1 -25427.731,E2 -25427.731} C_VEL
LIN {X 0,Y 149.98,Z 883.253,A -85,B 0,C 180,E1 -25430.303,E2 -25430.303} C_VEL
LIN {X 0,Y 146.071,Z 891.648,A -85,B 0,C 180,E1 -25433.008,E2 -25433.008} C_VEL
LIN {X 0,Y 141.884,Z 899.396,A -85,B 0,C 180,E1 -25436.114,E2 -25436.114} C_VEL
LIN {X 0,Y 137.281,Z 907.061,A -85,B 0,C 180,E1 -25440.121,E2 -25440.121} C_VEL
LIN {X 0,Y 133.688,Z 912.686,A -85,B 0,C 180,E1 -25444.001,E2 -25444.001} C_VEL
LIN {X 0,Y 129.769,Z 918.435,A -85,B 0,C 180,E1 -25449.368,E2 -25449.368} C_VEL
LIN {X 0,Y 126.88,Z 921.988,A -85,B 0,C 180,E1 -25453.901,E2 -25453.901} C_VEL
LIN {X 0,Y 125.453,Z 923.808,A -85,B 0,C 180,E1 -25457.03,E2 -25457.03} C_VEL
LIN {X 0,Y 123.838,Z 926.108,A -85,B 0,C 180,E1 -25463.461,E2 -25463.461} C_VEL
LIN {X 0,Y 123.14,Z 926.941,A -85,B 0,C 180,E1 -25469.978,E2 -25469.978} C_VEL
LIN {X 0,Y 123.826,Z 926.168,A -85,B 0,C 180,E1 -25476.496,E2 -25476.496} C_VEL
LIN {X 0,Y 125.418,Z 923.933,A -85,B 0,C 180,E1 -25482.93,E2 -25482.93} C_VEL
LIN {X 0,Y 127.717,Z 921.105,A -85,B 0,C 180,E1 -25487.594,E2 -25487.594} C_VEL
LIN {X 0,Y 130.675,Z 917.271,A -85,B 0,C 180,E1 -25492.092,E2 -25492.092} C_VEL
LIN {X 0,Y 134.37,Z 911.787,A -85,B 0,C 180,E1 -25496.893,E2 -25496.893} C_VEL
LIN {X 0,Y 138.732,Z 904.964,A -85,B 0,C 180,E1 -25501.257,E2 -25501.257} C_VEL
LIN {X 0,Y 143.459,Z 896.924,A -85,B 0,C 180,E1 -25505.118,E2 -25505.118} C_VEL
LIN {X 0,Y 147.687,Z 888.689,A -85,B 0,C 180,E1 -25508.19,E2 -25508.19} C_VEL
LIN {X 0,Y 152.197,Z 878.496,A -85,B 0,C 180,E1 -25511.122,E2 -25511.122} C_VEL
LIN {X 0,Y 156.226,Z 868.005,A -85,B 0,C 180,E1 -25513.405,E2 -25513.405} C_VEL
LIN {X 0,Y 159.749,Z 856.705,A -85,B 0,C 180,E1 -25515.303,E2 -25515.303} C_VEL
LIN {X 0,Y 162.661,Z 844.702,A -85,B 0,C 180,E1 -25516.783,E2 -25516.783} C_VEL
LIN {X 0,Y 164.576,Z 831.711,A -85,B 0,C 180,E1 -25518.041,E2 -25518.041} C_VEL
LIN {X 0,Y 165.637,Z 819.612,A -85,B 0,C 180,E1 -25518.798,E2 -25518.798} C_VEL
LIN {X 0,Y 166.681,Z 799.96,A -85,B 0,C 180,E1 -25519.675,E2 -25519.675} C_VEL
LIN {X 0,Y 161.586,Z 789.652,A -85,B 0,C 180,E1 -25522.685,E2 -25522.685} C_VEL
LIN {X 0,Y 156.539,Z 780.765,A -85,B 0,C 180,E1 -25526.003,E2 -25526.003} C_VEL
LIN {X 0,Y 151.586,Z 773.135,A -85,B 0,C 180,E1 -25529.722,E2 -25529.722} C_VEL
LIN {X 0,Y 148.452,Z 768.764,A -85,B 0,C 180,E1 -25532.414,E2 -25532.414} C_VEL
LIN {X 0,Y 145.931,Z 765.151,A -85,B 0,C 180,E1 -25534.887,E2 -25534.887} C_VEL
LIN {X 0,Y 143.296,Z 761.744,A -85,B 0,C 180,E1 -25537.816,E2 -25537.816} C_VEL
LIN {X 0,Y 142.418,Z 760.38,A -85,B 0,C 180,E1 -25538.941,E2 -25538.941} C_VEL
LIN {X 0,Y 140.009,Z 757.809,A -85,B 0,C 180,E1 -25542.283,E2 -25542.283} C_VEL
LIN {X 0,Y 138.768,Z 755.314,A -85,B 0,C 180,E1 -25544.579,E2 -25544.579} C_VEL
LIN {X 0,Y 135.98,Z 752.932,A -85,B 0,C 180,E1 -25551.08,E2 -25551.08} C_VEL
LIN {X 0,Y 135.076,Z 749.714,A -85,B 0,C 180,E1 -25558.509,E2 -25558.509} C_VEL
LIN {X 0,Y 135.118,Z 749.634,A -85,B 0,C 180,E1 -25560.372,E2 -25560.372} C_VEL
LIN {X 0,Y 135.633,Z 752.362,A -85,B 0,C 180,E1 -25565.575,E2 -25565.575} C_VEL
LIN {X 0,Y 137.91,Z 755.062,A -85,B 0,C 180,E1 -25571.948,E2 -25571.948} C_VEL
LIN {X 0,Y 139.751,Z 758.067,A -85,B 0,C 180,E1 -25575.449,E2 -25575.449} C_VEL
LIN {X 0,Y 144.222,Z 766.17,A -85,B 0,C 180,E1 -25581.719,E2 -25581.719} C_VEL
LIN {X 0,Y 148.088,Z 773.546,A -85,B 0,C 180,E1 -25585.85,E2 -25585.85} C_VEL
LIN {X 0,Y 151.276,Z 780.06,A -85,B 0,C 180,E1 -25588.763,E2 -25588.763} C_VEL
LIN {X 0,Y 154.083,Z 786.068,A -85,B 0,C 180,E1 -25591.063,E2 -25591.063} C_VEL
LIN {X 0,Y 157.466,Z 794.187,A -85,B 0,C 180,E1 -25593.623,E2 -25593.623} C_VEL
LIN {X 0,Y 161.292,Z 804.526,A -85,B 0,C 180,E1 -25596.297,E2 -25596.297} C_VEL
LIN {X 0,Y 162.15,Z 807.097,A -85,B 0,C 180,E1 -25596.876,E2 -25596.876} C_VEL
LIN {X 0,Y 162.796,Z 828.711,A -85,B 0,C 180,E1 -25598.655,E2 -25598.655} C_VEL
LIN {X 0,Y 163.031,Z 848.636,A -85,B 0,C 180,E1 -25600.081,E2 -25600.081} C_VEL
LIN {X 0,Y 161.59,Z 861.823,A -85,B 0,C 180,E1 -25600.733,E2 -25600.733} C_VEL
LIN {X 0,Y 158.962,Z 875.438,A -85,B 0,C 180,E1 -25601.778,E2 -25601.778} C_VEL
LIN {X 0,Y 155.995,Z 886.414,A -85,B 0,C 180,E1 -25602.966,E2 -25602.966} C_VEL
LIN {X 0,Y 151.921,Z 898.24,A -85,B 0,C 180,E1 -25604.692,E2 -25604.692} C_VEL
LIN {X 0,Y 146.941,Z 910.079,A -85,B 0,C 180,E1 -25607.063,E2 -25607.063} C_VEL
LIN {X 0,Y 141.714,Z 920.616,A -85,B 0,C 180,E1 -25609.884,E2 -25609.884} C_VEL
LIN {X 0,Y 137.025,Z 929.193,A -85,B 0,C 180,E1 -25612.967,E2 -25612.967} C_VEL
LIN {X 0,Y 132.02,Z 937.607,A -85,B 0,C 180,E1 -25616.958,E2 -25616.958} C_VEL
LIN {X 0,Y 128.552,Z 943.412,A -85,B 0,C 180,E1 -25620.552,E2 -25620.552} C_VEL
LIN {X 0,Y 125.164,Z 949.128,A -85,B 0,C 180,E1 -25625.12,E2 -25625.12} C_VEL
LIN {X 0,Y 122.744,Z 953.679,A -85,B 0,C 180,E1 -25629.932,E2 -25629.932} C_VEL
LIN {X 0,Y 121.324,Z 957.181,A -85,B 0,C 180,E1 -25634.914,E2 -25634.914} C_VEL
LIN {X 0,Y 120.909,Z 960.169,A -85,B 0,C 180,E1 -25641.17,E2 -25641.17} C_VEL
LIN {X 0,Y 121.513,Z 961.613,A -85,B 0,C 180,E1 -25646.707,E2 -25646.707} C_VEL
LIN {X 0,Y 122.016,Z 961.917,A -85,B 0,C 180,E1 -25650.022,E2 -25650.022} C_VEL
LIN {X 0,Y 121.506,Z 961.589,A -85,B 0,C 180,E1 -25653.338,E2 -25653.338} C_VEL
LIN {X 0,Y 120.975,Z 960.062,A -85,B 0,C 180,E1 -25659.029,E2 -25659.029} C_VEL
LIN {X 0,Y 121.671,Z 957.144,A -85,B 0,C 180,E1 -25665.088,E2 -25665.088} C_VEL
LIN {X 0,Y 123.378,Z 953.656,A -85,B 0,C 180,E1 -25670.007,E2 -25670.007} C_VEL
LIN {X 0,Y 125.987,Z 949.585,A -85,B 0,C 180,E1 -25674.289,E2 -25674.289} C_VEL
LIN {X 0,Y 126.607,Z 947.828,A -85,B 0,C 180,E1 -25675.927,E2 -25675.927} C_VEL
LIN {X 0,Y 126.159,Z 945.161,A -85,B 0,C 180,E1 -25678.788,E2 -25678.788} C_VEL
LIN {X 0,Y 125.872,Z 943.748,A -85,B 0,C 180,E1 -25681.171,E2 -25681.171} C_VEL
LIN {X 0,Y 126.567,Z 943.386,A -85,B 0,C 180,E1 -25683.103,E2 -25683.103} C_VEL
LIN {X 0,Y 126.92,Z 943.442,A -85,B 0,C 180,E1 -25683.525,E2 -25683.525} C_VEL
LIN {X 0,Y 133.716,Z 943.882,A -85,B 0,C 180,E1 -25689.125,E2 -25689.125} C_VEL
LIN {X 0,Y 142.019,Z 943.466,A -85,B 0,C 180,E1 -25693.875,E2 -25693.875} C_VEL
LIN {X 0,Y 151.635,Z 942.256,A -85,B 0,C 180,E1 -25697.887,E2 -25697.887} C_VEL
LIN {X 0,Y 156.894,Z 941.315,A -85,B 0,C 180,E1 -25699.619,E2 -25699.619} C_VEL
LIN {X 0,Y 157.338,Z 940.803,A -85,B 0,C 180,E1 -25700.528,E2 -25700.528} C_VEL
LIN {X 0,Y 151.152,Z 939.577,A -85,B 0,C 180,E1 -25702.811,E2 -25702.811} C_VEL
LIN {X 0,Y 141.888,Z 936.411,A -85,B 0,C 180,E1 -25706.985,E2 -25706.985} C_VEL
LIN {X 0,Y 133.688,Z 931.968,A -85,B 0,C 180,E1 -25711.762,E2 -25711.762} C_VEL
LIN {X 0,Y 126.874,Z 926.008,A -85,B 0,C 180,E1 -25717.185,E2 -25717.185} C_VEL
LIN {X 0,Y 121.725,Z 918.417,A -85,B 0,C 180,E1 -25723.221,E2 -25723.221} C_VEL
LIN {X 0,Y 118.951,Z 911.579,A -85,B 0,C 180,E1 -25728.066,E2 -25728.066} C_VEL
LIN {X 0,Y 116.953,Z 903.524,A -85,B 0,C 180,E1 -25733.097,E2 -25733.097} C_VEL
LIN {X 0,Y 115.987,Z 895.676,A -85,B 0,C 180,E1 -25737.395,E2 -25737.395} C_VEL
LIN {X 0,Y 115.632,Z 886.581,A -85,B 0,C 180,E1 -25741.742,E2 -25741.742} C_VEL
LIN {X 0,Y 115.993,Z 877.213,A -85,B 0,C 180,E1 -25745.651,E2 -25745.651} C_VEL
LIN {X 0,Y 116.458,Z 866.192,A -85,B 0,C 180,E1 -25749.443,E2 -25749.443} C_VEL
LIN {X 0,Y 116.322,Z 867.008,A -85,B 0,C 180,E1 -25750.443,E2 -25750.443} C_VEL
LIN {X 0,Y 117.186,Z 866.106,A -85,B 0,C 180,E1 -25752.117,E2 -25752.117} C_VEL
LIN {X 0,Y 118.626,Z 864.083,A -85,B 0,C 180,E1 -25753.709,E2 -25753.709} C_VEL
LIN {X 0,Y 121.606,Z 859.072,A -85,B 0,C 180,E1 -25755.89,E2 -25755.89} C_VEL
LIN {X 0,Y 122.799,Z 856.991,A -85,B 0,C 180,E1 -25756.628,E2 -25756.628} C_VEL
LIN {X 0,Y 124.008,Z 856.026,A -85,B 0,C 180,E1 -25758.162,E2 -25758.162} C_VEL
LIN {X 0,Y 125.638,Z 853.987,A -85,B 0,C 180,E1 -25759.611,E2 -25759.611} C_VEL
LIN {X 0,Y 128.267,Z 849.896,A -85,B 0,C 180,E1 -25761.289,E2 -25761.289} C_VEL
LIN {X 0,Y 131.205,Z 844.181,A -85,B 0,C 180,E1 -25762.748,E2 -25762.748} C_VEL
LIN {X 0,Y 134.92,Z 834.989,A -85,B 0,C 180,E1 -25764.321,E2 -25764.321} C_VEL
LIN {X 0,Y 137.124,Z 831.886,A -85,B 0,C 180,E1 -25765.827,E2 -25765.827} C_VEL
LIN {X 0,Y 139.466,Z 827.039,A -85,B 0,C 180,E1 -25767.167,E2 -25767.167} C_VEL
LIN {X 0,Y 142.423,Z 818.449,A -85,B 0,C 180,E1 -25768.557,E2 -25768.557} C_VEL
LIN {X 0,Y 146.215,Z 805.162,A -85,B 0,C 180,E1 -25769.991,E2 -25769.991} C_VEL
LIN {X 0,Y 147.253,Z 801.541,A -85,B 0,C 180,E1 -25770.361,E2 -25770.361} C_VEL
LIN {X 0,Y 149.926,Z 797.15,A -85,B 0,C 180,E1 -25771.729,E2 -25771.729} C_VEL
LIN {X 0,Y 152.755,Z 790.776,A -85,B 0,C 180,E1 -25772.921,E2 -25772.921} C_VEL
LIN {X 0,Y 153.935,Z 787.563,A -85,B 0,C 180,E1 -25773.346,E2 -25773.346} C_VEL
LIN {X 0,Y 154.814,Z 788.722,A -85,B 0,C 180,E1 -25773.953,E2 -25773.953} C_VEL
LIN {X 0,Y 159.889,Z 798.342,A -85,B 0,C 180,E1 -25777.384,E2 -25777.384} C_VEL
LIN {X 0,Y 161.862,Z 802.51,A -85,B 0,C 180,E1 -25778.62,E2 -25778.62} C_VEL
LIN {X 0,Y 160.386,Z 827.207,A -85,B 0,C 180,E1 -25779.852,E2 -25779.852} C_VEL
LIN {X 0,Y 158.596,Z 840.45,A -85,B 0,C 180,E1 -25780.903,E2 -25780.903} C_VEL
LIN {X 0,Y 156.034,Z 852.45,A -85,B 0,C 180,E1 -25782.242,E2 -25782.242} C_VEL
LIN {X 0,Y 152.762,Z 863.802,A -85,B 0,C 180,E1 -25783.957,E2 -25783.957} C_VEL
LIN {X 0,Y 148.542,Z 875.225,A -85,B 0,C 180,E1 -25786.194,E2 -25786.194} C_VEL
LIN {X 0,Y 144.165,Z 885.303,A -85,B 0,C 180,E1 -25788.822,E2 -25788.822} C_VEL
LIN {X 0,Y 139.619,Z 894.322,A -85,B 0,C 180,E1 -25791.908,E2 -25791.908} C_VEL
LIN {X 0,Y 134.427,Z 903.094,A -85,B 0,C 180,E1 -25795.783,E2 -25795.783} C_VEL
LIN {X 0,Y 129.388,Z 910.751,A -85,B 0,C 180,E1 -25800.352,E2 -25800.352} C_VEL
LIN {X 0,Y 125.402,Z 916.507,A -85,B 0,C 180,E1 -25805.123,E2 -25805.123} C_VEL
LIN {X 0,Y 123.217,Z 919.439,A -85,B 0,C 180,E1 -25808.217,E2 -25808.217} C_VEL
LIN {X 0,Y 120.144,Z 922.992,A -85,B 0,C 180,E1 -25812.971,E2 -25812.971} C_VEL
LIN {X 0,Y 118.615,Z 924.812,A -85,B 0,C 180,E1 -25816.268,E2 -25816.268} C_VEL
LIN {X 0,Y 116.859,Z 927.111,A -85,B 0,C 180,E1 -25823.069,E2 -25823.069} C_VEL
LIN {X 0,Y 116.112,Z 927.943,A -85,B 0,C 180,E1 -25829.977,E2 -25829.977} C_VEL
LIN {X 0,Y 116.846,Z 927.171,A -85,B 0,C 180,E1 -25836.886,E2 -25836.886} C_VEL
LIN {X 0,Y 118.578,Z 924.935,A -85,B 0,C 180,E1 -25843.69,E2 -25843.69} C_VEL
LIN {X 0,Y 121.036,Z 922.107,A -85,B 0,C 180,E1 -25848.6,E2 -25848.6} C_VEL
LIN {X 0,Y 124.191,Z 918.273,A -85,B 0,C 180,E1 -25853.311,E2 -25853.311} C_VEL
LIN {X 0,Y 128.141,Z 912.788,A -85,B 0,C 180,E1 -25858.314,E2 -25858.314} C_VEL
LIN {X 0,Y 132.774,Z 905.965,A -85,B 0,C 180,E1 -25862.831,E2 -25862.831} C_VEL
LIN {X 0,Y 137.77,Z 897.924,A -85,B 0,C 180,E1 -25866.8,E2 -25866.8} C_VEL
LIN {X 0,Y 142.23,Z 889.689,A -85,B 0,C 180,E1 -25869.941,E2 -25869.941} C_VEL
LIN {X 0,Y 146.975,Z 879.494,A -85,B 0,C 180,E1 -25872.925,E2 -25872.925} C_VEL
LIN {X 0,Y 151.198,Z 869.003,A -85,B 0,C 180,E1 -25875.235,E2 -25875.235} C_VEL
LIN {X 0,Y 154.886,Z 857.702,A -85,B 0,C 180,E1 -25877.152,E2 -25877.152} C_VEL
LIN {X 0,Y 157.929,Z 845.697,A -85,B 0,C 180,E1 -25878.643,E2 -25878.643} C_VEL
LIN {X 0,Y 160.027,Z 832.187,A -85,B 0,C 180,E1 -25879.956,E2 -25879.956} C_VEL
LIN {X 0,Y 161.176,Z 819.414,A -85,B 0,C 180,E1 -25880.736,E2 -25880.736} C_VEL
LIN {X 0,Y 162.056,Z 802.727,A -85,B 0,C 180,E1 -25881.517,E2 -25881.517} C_VEL
LIN {X 0,Y 157.304,Z 793.073,A -85,B 0,C 180,E1 -25884.591,E2 -25884.591} C_VEL
LIN {X 0,Y 153.375,Z 786.003,A -85,B 0,C 180,E1 -25887.407,E2 -25887.407} C_VEL
LIN {X 0,Y 149.057,Z 779.042,A -85,B 0,C 180,E1 -25890.906,E2 -25890.906} C_VEL
LIN {X 0,Y 146.236,Z 774.938,A -85,B 0,C 180,E1 -25893.505,E2 -25893.505} C_VEL
LIN {X 0,Y 143.828,Z 771.401,A -85,B 0,C 180,E1 -25896.035,E2 -25896.035} C_VEL
LIN {X 0,Y 141.121,Z 767.442,A -85,B 0,C 180,E1 -25899.36,E2 -25899.36} C_VEL
LIN {X 0,Y 138.261,Z 763.957,A -85,B 0,C 180,E1 -25903.66,E2 -25903.66} C_VEL
LIN {X 0,Y 137.374,Z 762.129,A -85,B 0,C 180,E1 -25905.463,E2 -25905.463} C_VEL
LIN {X 0,Y 134.174,Z 757.703,A -85,B 0,C 180,E1 -25916.997,E2 -25916.997} C_VEL
LIN {X 0,Y 134.233,Z 756.546,A -85,B 0,C 180,E1 -25919.25,E2 -25919.25} C_VEL
LIN {X 0,Y 134.219,Z 757.152,A -85,B 0,C 180,E1 -25920.75,E2 -25920.75} C_VEL
LIN {X 0,Y 134.984,Z 759.881,A -85,B 0,C 180,E1 -25926.54,E2 -25926.54} C_VEL
LIN {X 0,Y 136.676,Z 761.848,A -85,B 0,C 180,E1 -25931.237,E2 -25931.237} C_VEL
LIN {X 0,Y 138.225,Z 764.581,A -85,B 0,C 180,E1 -25934.445,E2 -25934.445} C_VEL
LIN {X 0,Y 142.197,Z 772.304,A -85,B 0,C 180,E1 -25940.526,E2 -25940.526} C_VEL
LIN {X 0,Y 145.573,Z 779.151,A -85,B 0,C 180,E1 -25944.46,E2 -25944.46} C_VEL
LIN {X 0,Y 148.673,Z 785.881,A -85,B 0,C 180,E1 -25947.54,E2 -25947.54} C_VEL
LIN {X 0,Y 151.919,Z 793.259,A -85,B 0,C 180,E1 -25950.38,E2 -25950.38} C_VEL
LIN {X 0,Y 156.244,Z 804.913,A -85,B 0,C 180,E1 -25953.823,E2 -25953.823} C_VEL
LIN {X 0,Y 157.892,Z 810.016,A -85,B 0,C 180,E1 -25955.063,E2 -25955.063} C_VEL
LIN {X 0,Y 158.415,Z 835.985,A -85,B 0,C 180,E1 -25957.227,E2 -25957.227} C_VEL
LIN {X 0,Y 158.361,Z 849.89,A -85,B 0,C 180,E1 -25958.21,E2 -25958.21} C_VEL
LIN {X 0,Y 156.598,Z 863.454,A -85,B 0,C 180,E1 -25958.932,E2 -25958.932} C_VEL
LIN {X 0,Y 154,Z 875.725,A -85,B 0,C 180,E1 -25959.923,E2 -25959.923} C_VEL
LIN {X 0,Y 150.619,Z 887.297,A -85,B 0,C 180,E1 -25961.232,E2 -25961.232} C_VEL
LIN {X 0,Y 146.413,Z 898.666,A -85,B 0,C 180,E1 -25962.975,E2 -25962.975} C_VEL
LIN {X 0,Y 141.833,Z 909.072,A -85,B 0,C 180,E1 -25965.112,E2 -25965.112} C_VEL
LIN {X 0,Y 136.355,Z 919.605,A -85,B 0,C 180,E1 -25967.96,E2 -25967.96} C_VEL
LIN {X 0,Y 131.381,Z 928.174,A -85,B 0,C 180,E1 -25971.087,E2 -25971.087} C_VEL
LIN {X 0,Y 126.077,Z 936.587,A -85,B 0,C 180,E1 -25975.183,E2 -25975.183} C_VEL
LIN {X 0,Y 121.276,Z 944.126,A -85,B 0,C 180,E1 -25980.192,E2 -25980.192} C_VEL
LIN {X 0,Y 117.689,Z 949.764,A -85,B 0,C 180,E1 -25985.317,E2 -25985.317} C_VEL
LIN {X 0,Y 115.387,Z 953.958,A -85,B 0,C 180,E1 -25990.454,E2 -25990.454} C_VEL
LIN {X 0,Y 114.104,Z 957.13,A -85,B 0,C 180,E1 -25995.762,E2 -25995.762} C_VEL
LIN {X 0,Y 113.849,Z 959.287,A -85,B 0,C 180,E1 -26001.002,E2 -26001.002} C_VEL
LIN {X 0,Y 114.428,Z 960.601,A -85,B 0,C 180,E1 -26006.502,E2 -26006.502} C_VEL
LIN {X 0,Y 114.948,Z 960.909,A -85,B 0,C 180,E1 -26010.023,E2 -26010.023} C_VEL
LIN {X 0,Y 114.426,Z 960.577,A -85,B 0,C 180,E1 -26013.544,E2 -26013.544} C_VEL
LIN {X 0,Y 113.957,Z 958.65,A -85,B 0,C 180,E1 -26020.685,E2 -26020.685} C_VEL
LIN {X 0,Y 114.785,Z 956.124,A -85,B 0,C 180,E1 -26026.016,E2 -26026.016} C_VEL
LIN {X 0,Y 116.705,Z 952.638,A -85,B 0,C 180,E1 -26031.204,E2 -26031.204} C_VEL
LIN {X 0,Y 119.899,Z 948.14,A -85,B 0,C 180,E1 -26036.103,E2 -26036.103} C_VEL
LIN {X 0,Y 124.181,Z 942.801,A -85,B 0,C 180,E1 -26040.408,E2 -26040.408} C_VEL
LIN {X 0,Y 126.92,Z 943.442,A -85,B 0,C 180,E1 -26043.525,E2 -26043.525} C_VEL
LIN {X 0,Y 128.858,Z 943.652,A -85,B 0,C 180,E1 -26046.026,E2 -26046.026} C_VEL
LIN {X 0,Y 131.293,Z 943.063,A -85,B 0,C 180,E1 -26050.254,E2 -26050.254} C_VEL
LIN {X 0,Y 134.677,Z 942.076,A -85,B 0,C 180,E1 -26054.229,E2 -26054.229} C_VEL
LIN {X 0,Y 137.992,Z 941.657,A -85,B 0,C 180,E1 -26056.262,E2 -26056.262} C_VEL
LIN {X 0,Y 147.058,Z 940.95,A -85,B 0,C 180,E1 -26059.9,E2 -26059.9} C_VEL
LIN {X 0,Y 145.558,Z 940.192,A -85,B 0,C 180,E1 -26061.121,E2 -26061.121} C_VEL
LIN {X 0,Y 135.975,Z 936.505,A -85,B 0,C 180,E1 -26065.351,E2 -26065.351} C_VEL
LIN {X 0,Y 129.484,Z 932.922,A -85,B 0,C 180,E1 -26068.96,E2 -26068.96} C_VEL
LIN {X 0,Y 122.002,Z 926.725,A -85,B 0,C 180,E1 -26074.403,E2 -26074.403} C_VEL
LIN {X 0,Y 117.474,Z 921.156,A -85,B 0,C 180,E1 -26078.964,E2 -26078.964} C_VEL
LIN {X 0,Y 113.554,Z 913.393,A -85,B 0,C 180,E1 -26084.75,E2 -26084.75} C_VEL
LIN {X 0,Y 111.394,Z 906.937,A -85,B 0,C 180,E1 -26089.09,E2 -26089.09} C_VEL
LIN {X 0,Y 109.692,Z 897.838,A -85,B 0,C 180,E1 -26094.485,E2 -26094.485} C_VEL
LIN {X 0,Y 108.978,Z 889.04,A -85,B 0,C 180,E1 -26099.076,E2 -26099.076} C_VEL
LIN {X 0,Y 108.966,Z 880.255,A -85,B 0,C 180,E1 -26103.12,E2 -26103.12} C_VEL
LIN {X 0,Y 108.726,Z 880.645,A -85,B 0,C 180,E1 -26103.706,E2 -26103.706} C_VEL
LIN {X 0,Y 109.907,Z 878.729,A -85,B 0,C 180,E1 -26107.348,E2 -26107.348} C_VEL
LIN {X 0,Y 112.1,Z 875.42,A -85,B 0,C 180,E1 -26109.928,E2 -26109.928} C_VEL
LIN {X 0,Y 113.1,Z 873.857,A -85,B 0,C 180,E1 -26110.744,E2 -26110.744} C_VEL
LIN {X 0,Y 115.227,Z 871.588,A -85,B 0,C 180,E1 -26114.121,E2 -26114.121} C_VEL
LIN {X 0,Y 117.818,Z 868.332,A -85,B 0,C 180,E1 -26116.461,E2 -26116.461} C_VEL
LIN {X 0,Y 121.27,Z 863.252,A -85,B 0,C 180,E1 -26118.587,E2 -26118.587} C_VEL
LIN {X 0,Y 123.969,Z 860.566,A -85,B 0,C 180,E1 -26120.972,E2 -26120.972} C_VEL
LIN {X 0,Y 126.835,Z 856.926,A -85,B 0,C 180,E1 -26122.823,E2 -26122.823} C_VEL
LIN {X 0,Y 130.614,Z 851.135,A -85,B 0,C 180,E1 -26124.646,E2 -26124.646} C_VEL
LIN {X 0,Y 134.88,Z 842.78,A -85,B 0,C 180,E1 -26126.185,E2 -26126.185} C_VEL
LIN {X 0,Y 136.3,Z 839.637,A -85,B 0,C 180,E1 -26126.716,E2 -26126.716} C_VEL
LIN {X 0,Y 139.266,Z 835.385,A -85,B 0,C 180,E1 -26128.339,E2 -26128.339} C_VEL
LIN {X 0,Y 142.241,Z 829.5,A -85,B 0,C 180,E1 -26129.683,E2 -26129.683} C_VEL
LIN {X 0,Y 145.492,Z 820.505,A -85,B 0,C 180,E1 -26130.992,E2 -26130.992} C_VEL
LIN {X 0,Y 149.973,Z 805.55,A -85,B 0,C 180,E1 -26132.522,E2 -26132.522} C_VEL
LIN {X 0,Y 153.205,Z 799.967,A -85,B 0,C 180,E1 -26133.974,E2 -26133.974} C_VEL
LIN {X 0,Y 153.497,Z 799.388,A -85,B 0,C 180,E1 -26134.093,E2 -26134.093} C_VEL
LIN {X 0,Y 154.449,Z 799.225,A -85,B 0,C 180,E1 -26134.619,E2 -26134.619} C_VEL
LIN {X 0,Y 157.436,Z 805.463,A -85,B 0,C 180,E1 -26136.702,E2 -26136.702} C_VEL
LIN {X 0,Y 155.968,Z 828.227,A -85,B 0,C 180,E1 -26137.866,E2 -26137.866} C_VEL
LIN {X 0,Y 154.147,Z 841.121,A -85,B 0,C 180,E1 -26138.897,E2 -26138.897} C_VEL
LIN {X 0,Y 151.399,Z 853.459,A -85,B 0,C 180,E1 -26140.272,E2 -26140.272} C_VEL
LIN {X 0,Y 148.001,Z 864.752,A -85,B 0,C 180,E1 -26141.993,E2 -26141.993} C_VEL
LIN {X 0,Y 143.552,Z 876.232,A -85,B 0,C 180,E1 -26144.252,E2 -26144.252} C_VEL
LIN {X 0,Y 138.952,Z 886.309,A -85,B 0,C 180,E1 -26146.914,E2 -26146.914} C_VEL
LIN {X 0,Y 134.158,Z 895.327,A -85,B 0,C 180,E1 -26150.056,E2 -26150.056} C_VEL
LIN {X 0,Y 128.676,Z 904.099,A -85,B 0,C 180,E1 -26154.023,E2 -26154.023} C_VEL
LIN {X 0,Y 123.33,Z 911.756,A -85,B 0,C 180,E1 -26158.736,E2 -26158.736} C_VEL
LIN {X 0,Y 119.063,Z 917.511,A -85,B 0,C 180,E1 -26163.7,E2 -26163.7} C_VEL
LIN {X 0,Y 116.72,Z 920.443,A -85,B 0,C 180,E1 -26166.936,E2 -26166.936} C_VEL
LIN {X 0,Y 113.443,Z 923.995,A -85,B 0,C 180,E1 -26171.932,E2 -26171.932} C_VEL
LIN {X 0,Y 111.8,Z 925.815,A -85,B 0,C 180,E1 -26175.413,E2 -26175.413} C_VEL
LIN {X 0,Y 109.885,Z 928.114,A -85,B 0,C 180,E1 -26182.627,E2 -26182.627} C_VEL
LIN {X 0,Y 109.084,Z 928.946,A -85,B 0,C 180,E1 -26189.976,E2 -26189.976} C_VEL
LIN {X 0,Y 109.872,Z 928.173,A -85,B 0,C 180,E1 -26197.325,E2 -26197.325} C_VEL
LIN {X 0,Y 111.761,Z 925.937,A -85,B 0,C 180,E1 -26204.543,E2 -26204.543} C_VEL
LIN {X 0,Y 114.397,Z 923.108,A -85,B 0,C 180,E1 -26209.722,E2 -26209.722} C_VEL
LIN {X 0,Y 117.769,Z 919.274,A -85,B 0,C 180,E1 -26214.665,E2 -26214.665} C_VEL
LIN {X 0,Y 122,Z 913.789,A -85,B 0,C 180,E1 -26219.88,E2 -26219.88} C_VEL
LIN {X 0,Y 126.926,Z 906.965,A -85,B 0,C 180,E1 -26224.551,E2 -26224.551} C_VEL
LIN {X 0,Y 132.209,Z 898.924,A -85,B 0,C 180,E1 -26228.624,E2 -26228.624} C_VEL
LIN {X 0,Y 136.916,Z 890.689,A -85,B 0,C 180,E1 -26231.829,E2 -26231.829} C_VEL
LIN {X 0,Y 141.909,Z 880.493,A -85,B 0,C 180,E1 -26234.858,E2 -26234.858} C_VEL
LIN {X 0,Y 146.333,Z 870.001,A -85,B 0,C 180,E1 -26237.189,E2 -26237.189} C_VEL
LIN {X 0,Y 150.195,Z 858.699,A -85,B 0,C 180,E1 -26239.118,E2 -26239.118} C_VEL
LIN {X 0,Y 153.376,Z 846.691,A -85,B 0,C 180,E1 -26240.614,E2 -26240.614} C_VEL
LIN {X 0,Y 155.544,Z 833.696,A -85,B 0,C 180,E1 -26241.887,E2 -26241.887} C_VEL
LIN {X 0,Y 156.728,Z 821.55,A -85,B 0,C 180,E1 -26242.673,E2 -26242.673} C_VEL
LIN {X 0,Y 157.632,Z 805.613,A -85,B 0,C 180,E1 -26243.444,E2 -26243.444} C_VEL
LIN {X 0,Y 153.211,Z 796.453,A -85,B 0,C 180,E1 -26246.601,E2 -26246.601} C_VEL
LIN {X 0,Y 148.78,Z 788.494,A -85,B 0,C 180,E1 -26250.167,E2 -26250.167} C_VEL
LIN {X 0,Y 144.798,Z 782.01,A -85,B 0,C 180,E1 -26253.903,E2 -26253.903} C_VEL
LIN {X 0,Y 141.803,Z 777.621,A -85,B 0,C 180,E1 -26257.202,E2 -26257.202} C_VEL
LIN {X 0,Y 139.095,Z 773.576,A -85,B 0,C 180,E1 -26260.827,E2 -26260.827} C_VEL
LIN {X 0,Y 136.665,Z 770.201,A -85,B 0,C 180,E1 -26264.934,E2 -26264.934} C_VEL
LIN {X 0,Y 136.105,Z 769,A -85,B 0,C 180,E1 -26266.183,E2 -26266.183} C_VEL
LIN {X 0,Y 133.345,Z 763.785,A -85,B 0,C 180,E1 -26279.245,E2 -26279.245} C_VEL
LIN {X 0,Y 134.741,Z 767.79,A -85,B 0,C 180,E1 -26288.624,E2 -26288.624} C_VEL
LIN {X 0,Y 135.593,Z 768.924,A -85,B 0,C 180,E1 -26290.85,E2 -26290.85} C_VEL
LIN {X 0,Y 136.806,Z 771.251,A -85,B 0,C 180,E1 -26293.555,E2 -26293.555} C_VEL
LIN {X 0,Y 140.294,Z 778.588,A -85,B 0,C 180,E1 -26299.383,E2 -26299.383} C_VEL
LIN {X 0,Y 143.293,Z 785.132,A -85,B 0,C 180,E1 -26303.198,E2 -26303.198} C_VEL
LIN {X 0,Y 145.934,Z 791.255,A -85,B 0,C 180,E1 -26306.069,E2 -26306.069} C_VEL
LIN {X 0,Y 148.833,Z 798.26,A -85,B 0,C 180,E1 -26308.852,E2 -26308.852} C_VEL
LIN {X 0,Y 152.899,Z 809.908,A -85,B 0,C 180,E1 -26312.397,E2 -26312.397} C_VEL
LIN {X 0,Y 153.808,Z 812.923,A -85,B 0,C 180,E1 -26313.154,E2 -26313.154} C_VEL
LIN {X 0,Y 154.074,Z 840.403,A -85,B 0,C 180,E1 -26315.467,E2 -26315.467} C_VEL
LIN {X 0,Y 153.902,Z 850.403,A -85,B 0,C 180,E1 -26316.188,E2 -26316.188} C_VEL
LIN {X 0,Y 151.998,Z 863.721,A -85,B 0,C 180,E1 -26316.926,E2 -26316.926} C_VEL
LIN {X 0,Y 149.207,Z 875.88,A -85,B 0,C 180,E1 -26317.945,E2 -26317.945} C_VEL
LIN {X 0,Y 145.392,Z 888.065,A -85,B 0,C 180,E1 -26319.373,E2 -26319.373} C_VEL
LIN {X 0,Y 141.046,Z 899.091,A -85,B 0,C 180,E1 -26321.126,E2 -26321.126} C_VEL
LIN {X 0,Y 136.298,Z 909.245,A -85,B 0,C 180,E1 -26323.286,E2 -26323.286} C_VEL
LIN {X 0,Y 131.169,Z 918.595,A -85,B 0,C 180,E1 -26325.883,E2 -26325.883} C_VEL
LIN {X 0,Y 125.903,Z 927.157,A -85,B 0,C 180,E1 -26329.044,E2 -26329.044} C_VEL
LIN {X 0,Y 120.279,Z 935.57,A -85,B 0,C 180,E1 -26333.239,E2 -26333.239} C_VEL
LIN {X 0,Y 116.3,Z 941.373,A -85,B 0,C 180,E1 -26337.082,E2 -26337.082} C_VEL
LIN {X 0,Y 112.346,Z 947.089,A -85,B 0,C 180,E1 -26342.048,E2 -26342.048} C_VEL
LIN {X 0,Y 109.404,Z 951.638,A -85,B 0,C 180,E1 -26347.357,E2 -26347.357} C_VEL
LIN {X 0,Y 107.526,Z 955.134,A -85,B 0,C 180,E1 -26352.922,E2 -26352.922} C_VEL
LIN {X 0,Y 106.799,Z 958.391,A -85,B 0,C 180,E1 -26360.782,E2 -26360.782} C_VEL
LIN {X 0,Y 107.321,Z 959.585,A -85,B 0,C 180,E1 -26366.27,E2 -26366.27} C_VEL
LIN {X 0,Y 107.877,Z 959.9,A -85,B 0,C 180,E1 -26370.025,E2 -26370.025} C_VEL
LIN {X 0,Y 107.325,Z 959.562,A -85,B 0,C 180,E1 -26373.779,E2 -26373.779} C_VEL
LIN {X 0,Y 106.943,Z 957.63,A -85,B 0,C 180,E1 -26381.395,E2 -26381.395} C_VEL
LIN {X 0,Y 107.954,Z 955.106,A -85,B 0,C 180,E1 -26387.06,E2 -26387.06} C_VEL
LIN {X 0,Y 110.095,Z 951.621,A -85,B 0,C 180,E1 -26392.545,E2 -26392.545} C_VEL
LIN {X 0,Y 113.587,Z 947.129,A -85,B 0,C 180,E1 -26397.673,E2 -26397.673} C_VEL
LIN {X 0,Y 118.312,Z 941.511,A -85,B 0,C 180,E1 -26402.342,E2 -26402.342} C_VEL
LIN {X 0,Y 119.433,Z 940.462,A -85,B 0,C 180,E1 -26403.153,E2 -26403.153} C_VEL
LIN {X 0,Y 124.773,Z 941.474,A -85,B 0,C 180,E1 -26408.31,E2 -26408.31} C_VEL
LIN {X 0,Y 132.655,Z 941.851,A -85,B 0,C 180,E1 -26413.554,E2 -26413.554} C_VEL
LIN {X 0,Y 137.992,Z 941.657,A -85,B 0,C 180,E1 -26416.262,E2 -26416.262} C_VEL
LIN {X 0,Y 138.925,Z 941.378,A -85,B 0,C 180,E1 -26417.153,E2 -26417.153} C_VEL
LIN {X 0,Y 138.721,Z 940.744,A -85,B 0,C 180,E1 -26418.408,E2 -26418.408} C_VEL
LIN {X 0,Y 137.553,Z 939.934,A -85,B 0,C 180,E1 -26419.649,E2 -26419.649} C_VEL
LIN {X 0,Y 135.061,Z 938.726,A -85,B 0,C 180,E1 -26421.15,E2 -26421.15} C_VEL
LIN {X 0,Y 129.013,Z 935.692,A -85,B 0,C 180,E1 -26424.153,E2 -26424.153} C_VEL
LIN {X 0,Y 119.401,Z 929.168,A -85,B 0,C 180,E1 -26429.979,E2 -26429.979} C_VEL
LIN {X 0,Y 112.427,Z 921.655,A -85,B 0,C 180,E1 -26436.026,E2 -26436.026} C_VEL
LIN {X 0,Y 108.495,Z 915.053,A -85,B 0,C 180,E1 -26441.102,E2 -26441.102} C_VEL
LIN {X 0,Y 105.498,Z 907.292,A -85,B 0,C 180,E1 -26446.517,E2 -26446.517} C_VEL
LIN {X 0,Y 103.685,Z 899.859,A -85,B 0,C 180,E1 -26451.228,E2 -26451.228} C_VEL
LIN {X 0,Y 102.672,Z 892.444,A -85,B 0,C 180,E1 -26455.461,E2 -26455.461} C_VEL
LIN {X 0,Y 102.339,Z 892.656,A -85,B 0,C 180,E1 -26456.062,E2 -26456.062} C_VEL
LIN {X 0,Y 102.425,Z 891.169,A -85,B 0,C 180,E1 -26460,E2 -26460} C_VEL
LIN {X 0,Y 103.843,Z 888.527,A -85,B 0,C 180,E1 -26462.91,E2 -26462.91} C_VEL
LIN {X 0,Y 104.558,Z 887.375,A -85,B 0,C 180,E1 -26463.854,E2 -26463.854} C_VEL
LIN {X 0,Y 105.469,Z 885.959,A -85,B 0,C 180,E1 -26465.737,E2 -26465.737} C_VEL
LIN {X 0,Y 106.773,Z 884.263,A -85,B 0,C 180,E1 -26468.996,E2 -26468.996} C_VEL
LIN {X 0,Y 108.594,Z 881.901,A -85,B 0,C 180,E1 -26471.196,E2 -26471.196} C_VEL
LIN {X 0,Y 110.547,Z 879.372,A -85,B 0,C 180,E1 -26472.857,E2 -26472.857} C_VEL
LIN {X 0,Y 113.142,Z 876.878,A -85,B 0,C 180,E1 -26476.234,E2 -26476.234} C_VEL
LIN {X 0,Y 115.965,Z 873.768,A -85,B 0,C 180,E1 -26478.553,E2 -26478.553} C_VEL
LIN {X 0,Y 119.576,Z 869.271,A -85,B 0,C 180,E1 -26480.649,E2 -26480.649} C_VEL
LIN {X 0,Y 124.668,Z 864.12,A -85,B 0,C 180,E1 -26484.124,E2 -26484.124} C_VEL
LIN {X 0,Y 128.445,Z 859.506,A -85,B 0,C 180,E1 -26485.959,E2 -26485.959} C_VEL
LIN {X 0,Y 132.228,Z 854.037,A -85,B 0,C 180,E1 -26487.418,E2 -26487.418} C_VEL
LIN {X 0,Y 137.709,Z 844.044,A -85,B 0,C 180,E1 -26489.065,E2 -26489.065} C_VEL
LIN {X 0,Y 141.223,Z 839.255,A -85,B 0,C 180,E1 -26490.67,E2 -26490.67} C_VEL
LIN {X 0,Y 144.565,Z 833.198,A -85,B 0,C 180,E1 -26491.917,E2 -26491.917} C_VEL
LIN {X 0,Y 148.299,Z 823.975,A -85,B 0,C 180,E1 -26493.153,E2 -26493.153} C_VEL
LIN {X 0,Y 152.818,Z 809.541,A -85,B 0,C 180,E1 -26494.556,E2 -26494.556} C_VEL
LIN {X 0,Y 153.236,Z 808.901,A -85,B 0,C 180,E1 -26494.738,E2 -26494.738} C_VEL
LIN {X 0,Y 151.745,Z 829.313,A -85,B 0,C 180,E1 -26495.774,E2 -26495.774} C_VEL
LIN {X 0,Y 149.784,Z 842.402,A -85,B 0,C 180,E1 -26496.83,E2 -26496.83} C_VEL
LIN {X 0,Y 146.954,Z 854.468,A -85,B 0,C 180,E1 -26498.181,E2 -26498.181} C_VEL
LIN {X 0,Y 143.444,Z 865.627,A -85,B 0,C 180,E1 -26499.883,E2 -26499.883} C_VEL
LIN {X 0,Y 138.739,Z 877.239,A -85,B 0,C 180,E1 -26502.172,E2 -26502.172} C_VEL
LIN {X 0,Y 133.906,Z 887.315,A -85,B 0,C 180,E1 -26504.859,E2 -26504.859} C_VEL
LIN {X 0,Y 128.849,Z 896.333,A -85,B 0,C 180,E1 -26508.05,E2 -26508.05} C_VEL
LIN {X 0,Y 123.058,Z 905.104,A -85,B 0,C 180,E1 -26512.1,E2 -26512.1} C_VEL
LIN {X 0,Y 117.379,Z 912.76,A -85,B 0,C 180,E1 -26516.956,E2 -26516.956} C_VEL
LIN {X 0,Y 112.806,Z 918.515,A -85,B 0,C 180,E1 -26522.118,E2 -26522.118} C_VEL
LIN {X 0,Y 110.288,Z 921.447,A -85,B 0,C 180,E1 -26525.506,E2 -26525.506} C_VEL
LIN {X 0,Y 106.784,Z 924.999,A -85,B 0,C 180,E1 -26530.762,E2 -26530.762} C_VEL
LIN {X 0,Y 105.013,Z 926.819,A -85,B 0,C 180,E1 -26534.447,E2 -26534.447} C_VEL
LIN {X 0,Y 102.919,Z 929.117,A -85,B 0,C 180,E1 -26542.125,E2 -26542.125} C_VEL
LIN {X 0,Y 102.056,Z 929.949,A -85,B 0,C 180,E1 -26549.974,E2 -26549.974} C_VEL
LIN {X 0,Y 102.905,Z 929.176,A -85,B 0,C 180,E1 -26557.824,E2 -26557.824} C_VEL
LIN {X 0,Y 104.973,Z 926.939,A -85,B 0,C 180,E1 -26565.506,E2 -26565.506} C_VEL
LIN {X 0,Y 107.808,Z 924.11,A -85,B 0,C 180,E1 -26570.983,E2 -26570.983} C_VEL
LIN {X 0,Y 111.421,Z 920.276,A -85,B 0,C 180,E1 -26576.173,E2 -26576.173} C_VEL
LIN {X 0,Y 115.959,Z 914.79,A -85,B 0,C 180,E1 -26581.61,E2 -26581.61} C_VEL
LIN {X 0,Y 121.203,Z 907.966,A -85,B 0,C 180,E1 -26586.436,E2 -26586.436} C_VEL
LIN {X 0,Y 126.795,Z 899.924,A -85,B 0,C 180,E1 -26590.607,E2 -26590.607} C_VEL
LIN {X 0,Y 131.762,Z 891.688,A -85,B 0,C 180,E1 -26593.868,E2 -26593.868} C_VEL
LIN {X 0,Y 137.017,Z 881.492,A -85,B 0,C 180,E1 -26596.931,E2 -26596.931} C_VEL
LIN {X 0,Y 141.651,Z 870.999,A -85,B 0,C 180,E1 -26599.275,E2 -26599.275} C_VEL
LIN {X 0,Y 145.692,Z 859.695,A -85,B 0,C 180,E1 -26601.208,E2 -26601.208} C_VEL
LIN {X 0,Y 149.01,Z 847.686,A -85,B 0,C 180,E1 -26602.705,E2 -26602.705} C_VEL
LIN {X 0,Y 151.302,Z 834.732,A -85,B 0,C 180,E1 -26603.977,E2 -26603.977} C_VEL
LIN {X 0,Y 152.587,Z 822.236,A -85,B 0,C 180,E1 -26604.791,E2 -26604.791} C_VEL
LIN {X 0,Y 153.404,Z 808.646,A -85,B 0,C 180,E1 -26605.463,E2 -26605.463} C_VEL
LIN {X 0,Y 149.213,Z 799.76,A -85,B 0,C 180,E1 -26608.794,E2 -26608.794} C_VEL
LIN {X 0,Y 145.103,Z 792.327,A -85,B 0,C 180,E1 -26612.504,E2 -26612.504} C_VEL
LIN {X 0,Y 141.971,Z 787.196,A -85,B 0,C 180,E1 -26615.798,E2 -26615.798} C_VEL
LIN {X 0,Y 139.913,Z 783.956,A -85,B 0,C 180,E1 -26618.304,E2 -26618.304} C_VEL
LIN {X 0,Y 137.64,Z 780.313,A -85,B 0,C 180,E1 -26621.582,E2 -26621.582} C_VEL
LIN {X 0,Y 135.261,Z 776.7,A -85,B 0,C 180,E1 -26625.951,E2 -26625.951} C_VEL
LIN {X 0,Y 134.732,Z 775.779,A -85,B 0,C 180,E1 -26627.191,E2 -26627.191} C_VEL
LIN {X 0,Y 132.416,Z 771.387,A -85,B 0,C 180,E1 -26638.479,E2 -26638.479} C_VEL
LIN {X 0,Y 132.439,Z 771.454,A -85,B 0,C 180,E1 -26640.38,E2 -26640.38} C_VEL
LIN {X 0,Y 134.009,Z 775.05,A -85,B 0,C 180,E1 -26649.052,E2 -26649.052} C_VEL
LIN {X 0,Y 135.27,Z 777.471,A -85,B 0,C 180,E1 -26652.28,E2 -26652.28} C_VEL
LIN {X 0,Y 138.337,Z 784.593,A -85,B 0,C 180,E1 -26658.034,E2 -26658.034} C_VEL
LIN {X 0,Y 140.987,Z 790.81,A -85,B 0,C 180,E1 -26661.762,E2 -26661.762} C_VEL
LIN {X 0,Y 144.448,Z 799.394,A -85,B 0,C 180,E1 -26665.785,E2 -26665.785} C_VEL
LIN {X 0,Y 147.532,Z 808.325,A -85,B 0,C 180,E1 -26668.935,E2 -26668.935} C_VEL
LIN {X 0,Y 149.89,Z 815.865,A -85,B 0,C 180,E1 -26671.138,E2 -26671.138} C_VEL
LIN {X 0,Y 149.865,Z 845.206,A -85,B 0,C 180,E1 -26673.627,E2 -26673.627} C_VEL
LIN {X 0,Y 149.397,Z 853.08,A -85,B 0,C 180,E1 -26674.165,E2 -26674.165} C_VEL
LIN {X 0,Y 146.996,Z 866.641,A -85,B 0,C 180,E1 -26675.011,E2 -26675.011} C_VEL
LIN {X 0,Y 144.013,Z 878.025,A -85,B 0,C 180,E1 -26676.044,E2 -26676.044} C_VEL
LIN {X 0,Y 139.702,Z 890.505,A -85,B 0,C 180,E1 -26677.632,E2 -26677.632} C_VEL
LIN {X 0,Y 134.581,Z 902.116,A -85,B 0,C 180,E1 -26679.658,E2 -26679.658} C_VEL
LIN {X 0,Y 129.071,Z 912.598,A -85,B 0,C 180,E1 -26682.143,E2 -26682.143} C_VEL
LIN {X 0,Y 123.866,Z 921.198,A -85,B 0,C 180,E1 -26684.862,E2 -26684.862} C_VEL
LIN {X 0,Y 117.553,Z 930.57,A -85,B 0,C 180,E1 -26688.913,E2 -26688.913} C_VEL
LIN {X 0,Y 111.996,Z 938.155,A -85,B 0,C 180,E1 -26693.438,E2 -26693.438} C_VEL
LIN {X 0,Y 107.402,Z 944.311,A -85,B 0,C 180,E1 -26698.465,E2 -26698.465} C_VEL
LIN {X 0,Y 103.772,Z 949.231,A -85,B 0,C 180,E1 -26703.913,E2 -26703.913} C_VEL
LIN {X 0,Y 101.286,Z 953.067,A -85,B 0,C 180,E1 -26709.729,E2 -26709.729} C_VEL
LIN {X 0,Y 100.256,Z 955.084,A -85,B 0,C 180,E1 -26713.745,E2 -26713.745} C_VEL
LIN {X 0,Y 99.761,Z 957.468,A -85,B 0,C 180,E1 -26720.498,E2 -26720.498} C_VEL
LIN {X 0,Y 100.201,Z 958.567,A -85,B 0,C 180,E1 -26726.005,E2 -26726.005} C_VEL
LIN {X 0,Y 100.801,Z 958.891,A -85,B 0,C 180,E1 -26730.026,E2 -26730.026} C_VEL
LIN {X 0,Y 100.212,Z 958.544,A -85,B 0,C 180,E1 -26734.048,E2 -26734.048} C_VEL
LIN {X 0,Y 99.976,Z 956.614,A -85,B 0,C 180,E1 -26742.201,E2 -26742.201} C_VEL
LIN {X 0,Y 101.171,Z 954.09,A -85,B 0,C 180,E1 -26748.242,E2 -26748.242} C_VEL
LIN {X 0,Y 103.561,Z 950.605,A -85,B 0,C 180,E1 -26754.054,E2 -26754.054} C_VEL
LIN {X 0,Y 107.375,Z 946.119,A -85,B 0,C 180,E1 -26759.426,E2 -26759.426} C_VEL
LIN {X 0,Y 112.429,Z 940.506,A -85,B 0,C 180,E1 -26764.262,E2 -26764.262} C_VEL
LIN {X 0,Y 114.927,Z 937.946,A -85,B 0,C 180,E1 -26766.013,E2 -26766.013} C_VEL
LIN {X 0,Y 123.512,Z 939.426,A -85,B 0,C 180,E1 -26773.09,E2 -26773.09} C_VEL
LIN {X 0,Y 132.965,Z 939.753,A -85,B 0,C 180,E1 -26778.211,E2 -26778.211} C_VEL
LIN {X 0,Y 137.425,Z 939.646,A -85,B 0,C 180,E1 -26780.12,E2 -26780.12} C_VEL
LIN {X 0,Y 135.008,Z 938.612,A -85,B 0,C 180,E1 -26781.342,E2 -26781.342} C_VEL
LIN {X 0,Y 129.013,Z 935.692,A -85,B 0,C 180,E1 -26784.153,E2 -26784.153} C_VEL
LIN {X 0,Y 124.974,Z 933.638,A -85,B 0,C 180,E1 -26785.859,E2 -26785.859} C_VEL
LIN {X 0,Y 117.529,Z 929.586,A -85,B 0,C 180,E1 -26788.28,E2 -26788.28} C_VEL
LIN {X 0,Y 110.619,Z 924.938,A -85,B 0,C 180,E1 -26790.953,E2 -26790.953} C_VEL
LIN {X 0,Y 107.539,Z 921.818,A -85,B 0,C 180,E1 -26793.066,E2 -26793.066} C_VEL
LIN {X 0,Y 102.654,Z 914.146,A -85,B 0,C 180,E1 -26798.935,E2 -26798.935} C_VEL
LIN {X 0,Y 99.349,Z 906.135,A -85,B 0,C 180,E1 -26804.617,E2 -26804.617} C_VEL
LIN {X 0,Y 98.264,Z 903.128,A -85,B 0,C 180,E1 -26806.822,E2 -26806.822} C_VEL
LIN {X 0,Y 97.81,Z 903.141,A -85,B 0,C 180,E1 -26807.552,E2 -26807.552} C_VEL
LIN {X 0,Y 96.884,Z 901.71,A -85,B 0,C 180,E1 -26811.658,E2 -26811.658} C_VEL
LIN {X 0,Y 97.795,Z 898.657,A -85,B 0,C 180,E1 -26815.879,E2 -26815.879} C_VEL
LIN {X 0,Y 98.482,Z 896.109,A -85,B 0,C 180,E1 -26821.836,E2 -26821.836} C_VEL
LIN {X 0,Y 100.276,Z 893.368,A -85,B 0,C 180,E1 -26825.026,E2 -26825.026} C_VEL
LIN {X 0,Y 101.067,Z 892.282,A -85,B 0,C 180,E1 -26825.987,E2 -26825.987} C_VEL
LIN {X 0,Y 104.138,Z 888.796,A -85,B 0,C 180,E1 -26831.681,E2 -26831.681} C_VEL
LIN {X 0,Y 106.823,Z 885.784,A -85,B 0,C 180,E1 -26834.284,E2 -26834.284} C_VEL
LIN {X 0,Y 107.918,Z 884.545,A -85,B 0,C 180,E1 -26835.1,E2 -26835.1} C_VEL
LIN {X 0,Y 111.463,Z 881.483,A -85,B 0,C 180,E1 -26838.892,E2 -26838.892} C_VEL
LIN {X 0,Y 115.197,Z 877.785,A -85,B 0,C 180,E1 -26841.473,E2 -26841.473} C_VEL
LIN {X 0,Y 118.8,Z 873.793,A -85,B 0,C 180,E1 -26843.286,E2 -26843.286} C_VEL
LIN {X 0,Y 123.516,Z 869.577,A -85,B 0,C 180,E1 -26846.166,E2 -26846.166} C_VEL
LIN {X 0,Y 127.262,Z 865.591,A -85,B 0,C 180,E1 -26847.884,E2 -26847.884} C_VEL
LIN {X 0,Y 131.983,Z 859.729,A -85,B 0,C 180,E1 -26849.542,E2 -26849.542} C_VEL
LIN {X 0,Y 136.996,Z 852.12,A -85,B 0,C 180,E1 -26850.865,E2 -26850.865} C_VEL
LIN {X 0,Y 138.75,Z 849.001,A -85,B 0,C 180,E1 -26851.279,E2 -26851.279} C_VEL
LIN {X 0,Y 144.17,Z 841.643,A -85,B 0,C 180,E1 -26853.259,E2 -26853.259} C_VEL
LIN {X 0,Y 146.747,Z 837.258,A -85,B 0,C 180,E1 -26854.043,E2 -26854.043} C_VEL
LIN {X 0,Y 144.257,Z 849.866,A -85,B 0,C 180,E1 -26855.3,E2 -26855.3} C_VEL
LIN {X 0,Y 140.645,Z 862.017,A -85,B 0,C 180,E1 -26856.89,E2 -26856.89} C_VEL
LIN {X 0,Y 136.341,Z 873.316,A -85,B 0,C 180,E1 -26858.892,E2 -26858.892} C_VEL
LIN {X 0,Y 131.849,Z 882.981,A -85,B 0,C 180,E1 -26861.131,E2 -26861.131} C_VEL
LIN {X 0,Y 126.875,Z 892.155,A -85,B 0,C 180,E1 -26863.91,E2 -26863.91} C_VEL
LIN {X 0,Y 121.615,Z 900.506,A -85,B 0,C 180,E1 -26867.207,E2 -26867.207} C_VEL
LIN {X 0,Y 115.685,Z 908.621,A -85,B 0,C 180,E1 -26871.46,E2 -26871.46} C_VEL
LIN {X 0,Y 110.123,Z 915.47,A -85,B 0,C 180,E1 -26876.402,E2 -26876.402} C_VEL
LIN {X 0,Y 105.207,Z 921.076,A -85,B 0,C 180,E1 -26882.094,E2 -26882.094} C_VEL
LIN {X 0,Y 101.314,Z 924.958,A -85,B 0,C 180,E1 -26887.545,E2 -26887.545} C_VEL
LIN {X 0,Y 98.26,Z 927.822,A -85,B 0,C 180,E1 -26893.348,E2 -26893.348} C_VEL
LIN {X 0,Y 95.962,Z 930.12,A -85,B 0,C 180,E1 -26901.55,E2 -26901.55} C_VEL
LIN {X 0,Y 95.028,Z 930.952,A -85,B 0,C 180,E1 -26909.972,E2 -26909.972} C_VEL
LIN {X 0,Y 95.947,Z 930.178,A -85,B 0,C 180,E1 -26918.395,E2 -26918.395} C_VEL
LIN {X 0,Y 98.218,Z 927.941,A -85,B 0,C 180,E1 -26926.602,E2 -26926.602} C_VEL
LIN {X 0,Y 101.277,Z 925.112,A -85,B 0,C 180,E1 -26932.407,E2 -26932.407} C_VEL
LIN {X 0,Y 105.159,Z 921.277,A -85,B 0,C 180,E1 -26937.862,E2 -26937.862} C_VEL
LIN {X 0,Y 110.035,Z 915.791,A -85,B 0,C 180,E1 -26943.529,E2 -26943.529} C_VEL
LIN {X 0,Y 115.624,Z 908.966,A -85,B 0,C 180,E1 -26948.505,E2 -26948.505} C_VEL
LIN {X 0,Y 121.546,Z 900.924,A -85,B 0,C 180,E1 -26952.764,E2 -26952.764} C_VEL
LIN {X 0,Y 126.789,Z 892.688,A -85,B 0,C 180,E1 -26956.07,E2 -26956.07} C_VEL
LIN {X 0,Y 132.317,Z 882.491,A -85,B 0,C 180,E1 -26959.155,E2 -26959.155} C_VEL
LIN {X 0,Y 137.169,Z 871.997,A -85,B 0,C 180,E1 -26961.5,E2 -26961.5} C_VEL
LIN {X 0,Y 141.395,Z 860.692,A -85,B 0,C 180,E1 -26963.428,E2 -26963.428} C_VEL
LIN {X 0,Y 144.862,Z 848.68,A -85,B 0,C 180,E1 -26964.916,E2 -26964.916} C_VEL
LIN {X 0,Y 147.302,Z 835.522,A -85,B 0,C 180,E1 -26966.21,E2 -26966.21} C_VEL
LIN {X 0,Y 148.657,Z 823.048,A -85,B 0,C 180,E1 -26967.016,E2 -26967.016} C_VEL
LIN {X 0,Y 149.331,Z 811.631,A -85,B 0,C 180,E1 -26967.626,E2 -26967.626} C_VEL
LIN {X 0,Y 145.763,Z 803.959,A -85,B 0,C 180,E1 -26970.779,E2 -26970.779} C_VEL
LIN {X 0,Y 142.193,Z 797.207,A -85,B 0,C 180,E1 -26974.375,E2 -26974.375} C_VEL
LIN {X 0,Y 138.61,Z 790.967,A -85,B 0,C 180,E1 -26978.727,E2 -26978.727} C_VEL
LIN {X 0,Y 135.921,Z 786.693,A -85,B 0,C 180,E1 -26982.83,E2 -26982.83} C_VEL
LIN {X 0,Y 133.783,Z 782.959,A -85,B 0,C 180,E1 -26987.292,E2 -26987.292} C_VEL
LIN {X 0,Y 131.539,Z 778.537,A -85,B 0,C 180,E1 -26998.469,E2 -26998.469} C_VEL
LIN {X 0,Y 131.552,Z 778.639,A -85,B 0,C 180,E1 -27000.287,E2 -27000.287} C_VEL
LIN {X 0,Y 133.194,Z 782.419,A -85,B 0,C 180,E1 -27009.299,E2 -27009.299} C_VEL
LIN {X 0,Y 133.962,Z 784.292,A -85,B 0,C 180,E1 -27011.442,E2 -27011.442} C_VEL
LIN {X 0,Y 136.562,Z 790.861,A -85,B 0,C 180,E1 -27016.827,E2 -27016.827} C_VEL
LIN {X 0,Y 138.768,Z 796.522,A -85,B 0,C 180,E1 -27020.28,E2 -27020.28} C_VEL
LIN {X 0,Y 141.753,Z 804.525,A -85,B 0,C 180,E1 -27024.144,E2 -27024.144} C_VEL
LIN {X 0,Y 144.926,Z 814.523,A -85,B 0,C 180,E1 -27027.725,E2 -27027.725} C_VEL
LIN {X 0,Y 146.184,Z 819.131,A -85,B 0,C 180,E1 -27029.059,E2 -27029.059} C_VEL
LIN {X 0,Y 145.776,Z 848.241,A -85,B 0,C 180,E1 -27031.549,E2 -27031.549} C_VEL
LIN {X 0,Y 145.171,Z 854.308,A -85,B 0,C 180,E1 -27031.945,E2 -27031.945} C_VEL
LIN {X 0,Y 142.564,Z 867.714,A -85,B 0,C 180,E1 -27032.838,E2 -27032.838} C_VEL
LIN {X 0,Y 138.973,Z 879.874,A -85,B 0,C 180,E1 -27033.977,E2 -27033.977} C_VEL
LIN {X 0,Y 134.801,Z 891.087,A -85,B 0,C 180,E1 -27035.489,E2 -27035.489} C_VEL
LIN {X 0,Y 129.503,Z 902.406,A -85,B 0,C 180,E1 -27037.508,E2 -27037.508} C_VEL
LIN {X 0,Y 124.418,Z 911.589,A -85,B 0,C 180,E1 -27039.718,E2 -27039.718} C_VEL
LIN {X 0,Y 118.948,Z 920.184,A -85,B 0,C 180,E1 -27042.429,E2 -27042.429} C_VEL
LIN {X 0,Y 113.344,Z 928.157,A -85,B 0,C 180,E1 -27045.805,E2 -27045.805} C_VEL
LIN {X 0,Y 107.253,Z 935.985,A -85,B 0,C 180,E1 -27050.326,E2 -27050.326} C_VEL
LIN {X 0,Y 101.368,Z 943.291,A -85,B 0,C 180,E1 -27056.348,E2 -27056.348} C_VEL
LIN {X 0,Y 97.392,Z 948.21,A -85,B 0,C 180,E1 -27062.06,E2 -27062.06} C_VEL
LIN {X 0,Y 94.582,Z 952.043,A -85,B 0,C 180,E1 -27068.222,E2 -27068.222} C_VEL
LIN {X 0,Y 93.404,Z 954.063,A -85,B 0,C 180,E1 -27072.515,E2 -27072.515} C_VEL
LIN {X 0,Y 92.722,Z 956.788,A -85,B 0,C 180,E1 -27081.31,E2 -27081.31} C_VEL
LIN {X 0,Y 93.086,Z 957.55,A -85,B 0,C 180,E1 -27085.699,E2 -27085.699} C_VEL
LIN {X 0,Y 93.718,Z 957.88,A -85,B 0,C 180,E1 -27090.028,E2 -27090.028} C_VEL
LIN {X 0,Y 93.105,Z 957.527,A -85,B 0,C 180,E1 -27094.358,E2 -27094.358} C_VEL
LIN {X 0,Y 93.028,Z 955.597,A -85,B 0,C 180,E1 -27103.128,E2 -27103.128} C_VEL
LIN {X 0,Y 94.405,Z 953.069,A -85,B 0,C 180,E1 -27109.601,E2 -27109.601} C_VEL
LIN {X 0,Y 97.114,Z 949.59,A -85,B 0,C 180,E1 -27115.764,E2 -27115.764} C_VEL
LIN {X 0,Y 101.278,Z 945.11,A -85,B 0,C 180,E1 -27121.391,E2 -27121.391} C_VEL
LIN {X 0,Y 106.686,Z 939.5,A -85,B 0,C 180,E1 -27126.39,E2 -27126.39} C_VEL
LIN {X 0,Y 111.069,Z 935.312,A -85,B 0,C 180,E1 -27129.282,E2 -27129.282} C_VEL
LIN {X 0,Y 115.754,Z 936.408,A -85,B 0,C 180,E1 -27133.233,E2 -27133.233} C_VEL
LIN {X 0,Y 126.485,Z 937.513,A -85,B 0,C 180,E1 -27139.509,E2 -27139.509} C_VEL
LIN {X 0,Y 127.498,Z 937.394,A -85,B 0,C 180,E1 -27140.251,E2 -27140.251} C_VEL
LIN {X 0,Y 117.577,Z 931.455,A -85,B 0,C 180,E1 -27145.4,E2 -27145.4} C_VEL
LIN {X 0,Y 109.514,Z 924.18,A -85,B 0,C 180,E1 -27151.229,E2 -27151.229} C_VEL
LIN {X 0,Y 107.539,Z 921.818,A -85,B 0,C 180,E1 -27153.066,E2 -27153.066} C_VEL
LIN {X 0,Y 105.376,Z 919.66,A -85,B 0,C 180,E1 -27154.49,E2 -27154.49} C_VEL
LIN {X 0,Y 100.594,Z 915.99,A -85,B 0,C 180,E1 -27156.358,E2 -27156.358} C_VEL
LIN {X 0,Y 96.054,Z 912.961,A -85,B 0,C 180,E1 -27158.606,E2 -27158.606} C_VEL
LIN {X 0,Y 94.342,Z 911.727,A -85,B 0,C 180,E1 -27160.585,E2 -27160.585} C_VEL
LIN {X 0,Y 93.564,Z 910.996,A -85,B 0,C 180,E1 -27162.515,E2 -27162.515} C_VEL
LIN {X 0,Y 93.198,Z 908.427,A -85,B 0,C 180,E1 -27166.925,E2 -27166.925} C_VEL
LIN {X 0,Y 92.07,Z 906.33,A -85,B 0,C 180,E1 -27173.105,E2 -27173.105} C_VEL
LIN {X 0,Y 93.17,Z 903.365,A -85,B 0,C 180,E1 -27177.839,E2 -27177.839} C_VEL
LIN {X 0,Y 93.773,Z 901.726,A -85,B 0,C 180,E1 -27181.929,E2 -27181.929} C_VEL
LIN {X 0,Y 94.598,Z 900.487,A -85,B 0,C 180,E1 -27184.261,E2 -27184.261} C_VEL
LIN {X 0,Y 97.44,Z 897.003,A -85,B 0,C 180,E1 -27188.294,E2 -27188.294} C_VEL
LIN {X 0,Y 99.638,Z 894.827,A -85,B 0,C 180,E1 -27192.217,E2 -27192.217} C_VEL
LIN {X 0,Y 102.974,Z 891.706,A -85,B 0,C 180,E1 -27195.843,E2 -27195.843} C_VEL
LIN {X 0,Y 105.207,Z 889.495,A -85,B 0,C 180,E1 -27197.494,E2 -27197.494} C_VEL
LIN {X 0,Y 108.359,Z 887.133,A -85,B 0,C 180,E1 -27200.638,E2 -27200.638} C_VEL
LIN {X 0,Y 113.238,Z 882.876,A -85,B 0,C 180,E1 -27203.792,E2 -27203.792} C_VEL
LIN {X 0,Y 118.65,Z 877.736,A -85,B 0,C 180,E1 -27206.374,E2 -27206.374} C_VEL
LIN {X 0,Y 122.155,Z 874.924,A -85,B 0,C 180,E1 -27208.278,E2 -27208.278} C_VEL
LIN {X 0,Y 126.377,Z 870.942,A -85,B 0,C 180,E1 -27210.034,E2 -27210.034} C_VEL
LIN {X 0,Y 132.618,Z 864.052,A -85,B 0,C 180,E1 -27211.984,E2 -27211.984} C_VEL
LIN {X 0,Y 137.851,Z 856.933,A -85,B 0,C 180,E1 -27213.157,E2 -27213.157} C_VEL
LIN {X 0,Y 138.857,Z 855.4,A -85,B 0,C 180,E1 -27213.358,E2 -27213.358} C_VEL
LIN {X 0,Y 137.561,Z 860.073,A -85,B 0,C 180,E1 -27214.101,E2 -27214.101} C_VEL
LIN {X 0,Y 133.475,Z 871.128,A -85,B 0,C 180,E1 -27215.913,E2 -27215.913} C_VEL
LIN {X 0,Y 128.538,Z 881.681,A -85,B 0,C 180,E1 -27218.161,E2 -27218.161} C_VEL
LIN {X 0,Y 123.221,Z 891.255,A -85,B 0,C 180,E1 -27220.883,E2 -27220.883} C_VEL
LIN {X 0,Y 117.672,Z 899.934,A -85,B 0,C 180,E1 -27224.188,E2 -27224.188} C_VEL
LIN {X 0,Y 111.29,Z 908.42,A -85,B 0,C 180,E1 -27228.436,E2 -27228.436} C_VEL
LIN {X 0,Y 105.485,Z 915.169,A -85,B 0,C 180,E1 -27233.128,E2 -27233.128} C_VEL
LIN {X 0,Y 100.596,Z 920.523,A -85,B 0,C 180,E1 -27238.372,E2 -27238.372} C_VEL
LIN {X 0,Y 97.671,Z 923.454,A -85,B 0,C 180,E1 -27242.085,E2 -27242.085} C_VEL
LIN {X 0,Y 93.627,Z 927.006,A -85,B 0,C 180,E1 -27247.927,E2 -27247.927} C_VEL
LIN {X 0,Y 91.548,Z 928.825,A -85,B 0,C 180,E1 -27252.088,E2 -27252.088} C_VEL
LIN {X 0,Y 89.017,Z 931.123,A -85,B 0,C 180,E1 -27260.885,E2 -27260.885} C_VEL
LIN {X 0,Y 88,Z 931.954,A -85,B 0,C 180,E1 -27269.97,E2 -27269.97} C_VEL
LIN {X 0,Y 89,Z 931.18,A -85,B 0,C 180,E1 -27279.056,E2 -27279.056} C_VEL
LIN {X 0,Y 91.504,Z 928.943,A -85,B 0,C 180,E1 -27287.86,E2 -27287.86} C_VEL
LIN {X 0,Y 94.818,Z 926.114,A -85,B 0,C 180,E1 -27294.026,E2 -27294.026} C_VEL
LIN {X 0,Y 99.001,Z 922.279,A -85,B 0,C 180,E1 -27299.763,E2 -27299.763} C_VEL
LIN {X 0,Y 104.249,Z 916.792,A -85,B 0,C 180,E1 -27305.663,E2 -27305.663} C_VEL
LIN {X 0,Y 110.211,Z 909.967,A -85,B 0,C 180,E1 -27310.78,E2 -27310.78} C_VEL
LIN {X 0,Y 116.484,Z 901.925,A -85,B 0,C 180,E1 -27315.112,E2 -27315.112} C_VEL
LIN {X 0,Y 122.018,Z 893.688,A -85,B 0,C 180,E1 -27318.447,E2 -27318.447} C_VEL
LIN {X 0,Y 127.831,Z 883.49,A -85,B 0,C 180,E1 -27321.539,E2 -27321.539} C_VEL
LIN {X 0,Y 132.908,Z 872.995,A -85,B 0,C 180,E1 -27323.872,E2 -27323.872} C_VEL
LIN {X 0,Y 137.324,Z 861.689,A -85,B 0,C 180,E1 -27325.784,E2 -27325.784} C_VEL
LIN {X 0,Y 140.937,Z 849.674,A -85,B 0,C 180,E1 -27327.256,E2 -27327.256} C_VEL
LIN {X 0,Y 143.499,Z 836.632,A -85,B 0,C 180,E1 -27328.529,E2 -27328.529} C_VEL
LIN {X 0,Y 144.879,Z 824.678,A -85,B 0,C 180,E1 -27329.322,E2 -27329.322} C_VEL
LIN {X 0,Y 145.542,Z 814.93,A -85,B 0,C 180,E1 -27329.834,E2 -27329.834} C_VEL
LIN {X 0,Y 142.655,Z 808.491,A -85,B 0,C 180,E1 -27332.69,E2 -27332.69} C_VEL
LIN {X 0,Y 139.302,Z 801.907,A -85,B 0,C 180,E1 -27336.482,E2 -27336.482} C_VEL
LIN {X 0,Y 136.415,Z 796.71,A -85,B 0,C 180,E1 -27340.435,E2 -27340.435} C_VEL
LIN {X 0,Y 134.518,Z 793.384,A -85,B 0,C 180,E1 -27343.654,E2 -27343.654} C_VEL
LIN {X 0,Y 132.366,Z 789.488,A -85,B 0,C 180,E1 -27348.612,E2 -27348.612} C_VEL
LIN {X 0,Y 130.66,Z 785.698,A -85,B 0,C 180,E1 -27358.459,E2 -27358.459} C_VEL
LIN {X 0,Y 130.666,Z 785.858,A -85,B 0,C 180,E1 -27360.289,E2 -27360.289} C_VEL
LIN {X 0,Y 132.118,Z 789.395,A -85,B 0,C 180,E1 -27368.797,E2 -27368.797} C_VEL
LIN {X 0,Y 132.688,Z 791.079,A -85,B 0,C 180,E1 -27370.587,E2 -27370.587} C_VEL
LIN {X 0,Y 134.847,Z 797.15,A -85,B 0,C 180,E1 -27375.589,E2 -27375.589} C_VEL
LIN {X 0,Y 136.683,Z 802.398,A -85,B 0,C 180,E1 -27378.818,E2 -27378.818} C_VEL
LIN {X 0,Y 139.246,Z 809.908,A -85,B 0,C 180,E1 -27382.536,E2 -27382.536} C_VEL
LIN {X 0,Y 142.108,Z 819.739,A -85,B 0,C 180,E1 -27386.148,E2 -27386.148} C_VEL
LIN {X 0,Y 142.658,Z 822.351,A -85,B 0,C 180,E1 -27386.853,E2 -27386.853} C_VEL
LIN {X 0,Y 141.978,Z 849.439,A -85,B 0,C 180,E1 -27389.221,E2 -27389.221} C_VEL
LIN {X 0,Y 140.801,Z 857.526,A -85,B 0,C 180,E1 -27389.726,E2 -27389.726} C_VEL
LIN {X 0,Y 137.891,Z 870.162,A -85,B 0,C 180,E1 -27390.653,E2 -27390.653} C_VEL
LIN {X 0,Y 133.883,Z 882.507,A -85,B 0,C 180,E1 -27391.918,E2 -27391.918} C_VEL
LIN {X 0,Y 128.73,Z 894.63,A -85,B 0,C 180,E1 -27393.68,E2 -27393.68} C_VEL
LIN {X 0,Y 123.304,Z 905.024,A -85,B 0,C 180,E1 -27395.73,E2 -27395.73} C_VEL
LIN {X 0,Y 116.805,Z 915.561,A -85,B 0,C 180,E1 -27398.58,E2 -27398.58} C_VEL
LIN {X 0,Y 110.633,Z 924.111,A -85,B 0,C 180,E1 -27401.759,E2 -27401.759} C_VEL
LIN {X 0,Y 103.908,Z 932.519,A -85,B 0,C 180,E1 -27406.149,E2 -27406.149} C_VEL
LIN {X 0,Y 98.043,Z 939.356,A -85,B 0,C 180,E1 -27411.193,E2 -27411.193} C_VEL
LIN {X 0,Y 92.449,Z 945.684,A -85,B 0,C 180,E1 -27417.887,E2 -27417.887} C_VEL
LIN {X 0,Y 88.879,Z 949.87,A -85,B 0,C 180,E1 -27424.256,E2 -27424.256} C_VEL
LIN {X 0,Y 86.578,Z 953.039,A -85,B 0,C 180,E1 -27431.087,E2 -27431.087} C_VEL
LIN {X 0,Y 85.668,Z 955.769,A -85,B 0,C 180,E1 -27440.589,E2 -27440.589} C_VEL
LIN {X 0,Y 85.98,Z 956.533,A -85,B 0,C 180,E1 -27445.343,E2 -27445.343} C_VEL
LIN {X 0,Y 86.628,Z 956.869,A -85,B 0,C 180,E1 -27450.031,E2 -27450.031} C_VEL
LIN {X 0,Y 86.005,Z 956.511,A -85,B 0,C 180,E1 -27454.718,E2 -27454.718} C_VEL
LIN {X 0,Y 86.1,Z 954.58,A -85,B 0,C 180,E1 -27464.206,E2 -27464.206} C_VEL
LIN {X 0,Y 87.706,Z 952.049,A -85,B 0,C 180,E1 -27471.168,E2 -27471.168} C_VEL
LIN {X 0,Y 90.771,Z 948.576,A -85,B 0,C 180,E1 -27477.712,E2 -27477.712} C_VEL
LIN {X 0,Y 95.305,Z 944.098,A -85,B 0,C 180,E1 -27483.609,E2 -27483.609} C_VEL
LIN {X 0,Y 101.107,Z 938.494,A -85,B 0,C 180,E1 -27488.757,E2 -27488.757} C_VEL
LIN {X 0,Y 107.341,Z 932.582,A -85,B 0,C 180,E1 -27492.542,E2 -27492.542} C_VEL
LIN {X 0,Y 116.141,Z 934.369,A -85,B 0,C 180,E1 -27498.735,E2 -27498.735} C_VEL
LIN {X 0,Y 117.983,Z 934.417,A -85,B 0,C 180,E1 -27500.02,E2 -27500.02} C_VEL
LIN {X 0,Y 107.453,Z 926.56,A -85,B 0,C 180,E1 -27506.224,E2 -27506.224} C_VEL
LIN {X 0,Y 99.955,Z 917.934,A -85,B 0,C 180,E1 -27512.805,E2 -27512.805} C_VEL
LIN {X 0,Y 96.603,Z 912.712,A -85,B 0,C 180,E1 -27516.981,E2 -27516.981} C_VEL
LIN {X 0,Y 95.38,Z 912.579,A -85,B 0,C 180,E1 -27518.382,E2 -27518.382} C_VEL
LIN {X 0,Y 94.342,Z 911.727,A -85,B 0,C 180,E1 -27520.585,E2 -27520.585} C_VEL
LIN {X 0,Y 93.014,Z 911.253,A -85,B 0,C 180,E1 -27522.875,E2 -27522.875} C_VEL
LIN {X 0,Y 87.629,Z 911.752,A -85,B 0,C 180,E1 -27530.696,E2 -27530.696} C_VEL
LIN {X 0,Y 87.104,Z 911.165,A -85,B 0,C 180,E1 -27533.244,E2 -27533.244} C_VEL
LIN {X 0,Y 87.2,Z 910.318,A -85,B 0,C 180,E1 -27535.377,E2 -27535.377} C_VEL
LIN {X 0,Y 88.406,Z 907.819,A -85,B 0,C 180,E1 -27540,E2 -27540} C_VEL
LIN {X 0,Y 89.505,Z 905.98,A -85,B 0,C 180,E1 -27544.504,E2 -27544.504} C_VEL
LIN {X 0,Y 90.522,Z 904.791,A -85,B 0,C 180,E1 -27546.688,E2 -27546.688} C_VEL
LIN {X 0,Y 93.679,Z 901.553,A -85,B 0,C 180,E1 -27550.808,E2 -27550.808} C_VEL
LIN {X 0,Y 98.053,Z 897.914,A -85,B 0,C 180,E1 -27556.661,E2 -27556.661} C_VEL
LIN {X 0,Y 101.241,Z 895.261,A -85,B 0,C 180,E1 -27559.253,E2 -27559.253} C_VEL
LIN {X 0,Y 102.441,Z 894.222,A -85,B 0,C 180,E1 -27560.062,E2 -27560.062} C_VEL
LIN {X 0,Y 106.28,Z 891.597,A -85,B 0,C 180,E1 -27563.376,E2 -27563.376} C_VEL
LIN {X 0,Y 111.957,Z 887.156,A -85,B 0,C 180,E1 -27566.597,E2 -27566.597} C_VEL
LIN {X 0,Y 117.043,Z 882.778,A -85,B 0,C 180,E1 -27568.71,E2 -27568.71} C_VEL
LIN {X 0,Y 122.293,Z 878.816,A -85,B 0,C 180,E1 -27571.146,E2 -27571.146} C_VEL
LIN {X 0,Y 128.392,Z 873.355,A -85,B 0,C 180,E1 -27573.188,E2 -27573.188} C_VEL
LIN {X 0,Y 128.247,Z 874.791,A -85,B 0,C 180,E1 -27573.895,E2 -27573.895} C_VEL
LIN {X 0,Y 123.06,Z 884.994,A -85,B 0,C 180,E1 -27576.195,E2 -27576.195} C_VEL
LIN {X 0,Y 117.564,Z 894.166,A -85,B 0,C 180,E1 -27578.969,E2 -27578.969} C_VEL
LIN {X 0,Y 111.71,Z 902.517,A -85,B 0,C 180,E1 -27582.303,E2 -27582.303} C_VEL
LIN {X 0,Y 105.057,Z 910.631,A -85,B 0,C 180,E1 -27586.678,E2 -27586.678} C_VEL
LIN {X 0,Y 98.723,Z 917.479,A -85,B 0,C 180,E1 -27591.883,E2 -27591.883} C_VEL
LIN {X 0,Y 93.018,Z 923.084,A -85,B 0,C 180,E1 -27598.038,E2 -27598.038} C_VEL
LIN {X 0,Y 88.487,Z 926.965,A -85,B 0,C 180,E1 -27604.066,E2 -27604.066} C_VEL
LIN {X 0,Y 84.888,Z 929.829,A -85,B 0,C 180,E1 -27610.629,E2 -27610.629} C_VEL
LIN {X 0,Y 82.085,Z 932.126,A -85,B 0,C 180,E1 -27620.108,E2 -27620.108} C_VEL
LIN {X 0,Y 80.972,Z 932.957,A -85,B 0,C 180,E1 -27629.967,E2 -27629.967} C_VEL
LIN {X 0,Y 82.067,Z 932.183,A -85,B 0,C 180,E1 -27639.828,E2 -27639.828} C_VEL
LIN {X 0,Y 84.842,Z 929.945,A -85,B 0,C 180,E1 -27649.316,E2 -27649.316} C_VEL
LIN {X 0,Y 88.445,Z 927.115,A -85,B 0,C 180,E1 -27655.88,E2 -27655.88} C_VEL
LIN {X 0,Y 92.965,Z 923.28,A -85,B 0,C 180,E1 -27661.914,E2 -27661.914} C_VEL
LIN {X 0,Y 98.624,Z 917.793,A -85,B 0,C 180,E1 -27668.044,E2 -27668.044} C_VEL
LIN {X 0,Y 104.99,Z 910.968,A -85,B 0,C 180,E1 -27673.286,E2 -27673.286} C_VEL
LIN {X 0,Y 111.635,Z 902.925,A -85,B 0,C 180,E1 -27677.668,E2 -27677.668} C_VEL
LIN {X 0,Y 117.473,Z 894.687,A -85,B 0,C 180,E1 -27681.013,E2 -27681.013} C_VEL
LIN {X 0,Y 123.582,Z 884.489,A -85,B 0,C 180,E1 -27684.091,E2 -27684.091} C_VEL
LIN {X 0,Y 128.89,Z 873.993,A -85,B 0,C 180,E1 -27686.397,E2 -27686.397} C_VEL
LIN {X 0,Y 133.698,Z 862.146,A -85,B 0,C 180,E1 -27688.353,E2 -27688.353} C_VEL
LIN {X 0,Y 137.528,Z 849.517,A -85,B 0,C 180,E1 -27689.863,E2 -27689.863} C_VEL
LIN {X 0,Y 140.181,Z 836.254,A -85,B 0,C 180,E1 -27691.1,E2 -27691.1} C_VEL
LIN {X 0,Y 141.49,Z 824.969,A -85,B 0,C 180,E1 -27691.807,E2 -27691.807} C_VEL
LIN {X 0,Y 141.97,Z 818.247,A -85,B 0,C 180,E1 -27692.164,E2 -27692.164} C_VEL
LIN {X 0,Y 138.975,Z 811.447,A -85,B 0,C 180,E1 -27695.566,E2 -27695.566} C_VEL
LIN {X 0,Y 136.037,Z 805.586,A -85,B 0,C 180,E1 -27699.492,E2 -27699.492} C_VEL
LIN {X 0,Y 134.124,Z 802.024,A -85,B 0,C 180,E1 -27702.593,E2 -27702.593} C_VEL
LIN {X 0,Y 132.867,Z 799.646,A -85,B 0,C 180,E1 -27705.057,E2 -27705.057} C_VEL
LIN {X 0,Y 131.264,Z 796.39,A -85,B 0,C 180,E1 -27709.199,E2 -27709.199} C_VEL
LIN {X 0,Y 129.78,Z 792.863,A -85,B 0,C 180,E1 -27718.448,E2 -27718.448} C_VEL
LIN {X 0,Y 129.788,Z 793.142,A -85,B 0,C 180,E1 -27720.582,E2 -27720.582} C_VEL
LIN {X 0,Y 131.054,Z 796.368,A -85,B 0,C 180,E1 -27728.286,E2 -27728.286} C_VEL
LIN {X 0,Y 133.159,Z 803.266,A -85,B 0,C 180,E1 -27734.226,E2 -27734.226} C_VEL
LIN {X 0,Y 134.723,Z 808.275,A -85,B 0,C 180,E1 -27737.357,E2 -27737.357} C_VEL
LIN {X 0,Y 136.969,Z 815.714,A -85,B 0,C 180,E1 -27741.05,E2 -27741.05} C_VEL
LIN {X 0,Y 139.267,Z 824.56,A -85,B 0,C 180,E1 -27744.345,E2 -27744.345} C_VEL
LIN {X 0,Y 139.167,Z 831.635,A -85,B 0,C 180,E1 -27745.084,E2 -27745.084} C_VEL
LIN {X 0,Y 138.4,Z 850.037,A -85,B 0,C 180,E1 -27746.725,E2 -27746.725} C_VEL
LIN {X 0,Y 137.218,Z 857.51,A -85,B 0,C 180,E1 -27747.207,E2 -27747.207} C_VEL
LIN {X 0,Y 134.267,Z 869.658,A -85,B 0,C 180,E1 -27748.088,E2 -27748.088} C_VEL
LIN {X 0,Y 129.986,Z 882.174,A -85,B 0,C 180,E1 -27749.342,E2 -27749.342} C_VEL
LIN {X 0,Y 124.936,Z 893.622,A -85,B 0,C 180,E1 -27750.972,E2 -27750.972} C_VEL
LIN {X 0,Y 118.592,Z 905.196,A -85,B 0,C 180,E1 -27753.215,E2 -27753.215} C_VEL
LIN {X 0,Y 112.493,Z 914.546,A -85,B 0,C 180,E1 -27755.737,E2 -27755.737} C_VEL
LIN {X 0,Y 106.026,Z 923.098,A -85,B 0,C 180,E1 -27758.889,E2 -27758.889} C_VEL
LIN {X 0,Y 98.898,Z 931.505,A -85,B 0,C 180,E1 -27763.291,E2 -27763.291} C_VEL
LIN {X 0,Y 92.571,Z 938.336,A -85,B 0,C 180,E1 -27768.413,E2 -27768.413} C_VEL
LIN {X 0,Y 86.479,Z 944.665,A -85,B 0,C 180,E1 -27775.368,E2 -27775.368} C_VEL
LIN {X 0,Y 82.473,Z 948.847,A -85,B 0,C 180,E1 -27782.09,E2 -27782.09} C_VEL
LIN {X 0,Y 79.837,Z 952.018,A -85,B 0,C 180,E1 -27789.42,E2 -27789.42} C_VEL
LIN {X 0,Y 78.615,Z 954.748,A -85,B 0,C 180,E1 -27799.736,E2 -27799.736} C_VEL
LIN {X 0,Y 78.879,Z 955.517,A -85,B 0,C 180,E1 -27804.923,E2 -27804.923} C_VEL
LIN {X 0,Y 79.534,Z 955.856,A -85,B 0,C 180,E1 -27810.034,E2 -27810.034} C_VEL
LIN {X 0,Y 78.914,Z 955.496,A -85,B 0,C 180,E1 -27815.143,E2 -27815.143} C_VEL
LIN {X 0,Y 79.199,Z 953.561,A -85,B 0,C 180,E1 -27825.473,E2 -27825.473} C_VEL
LIN {X 0,Y 81.093,Z 951.03,A -85,B 0,C 180,E1 -27832.988,E2 -27832.988} C_VEL
LIN {X 0,Y 84.547,Z 947.562,A -85,B 0,C 180,E1 -27839.951,E2 -27839.951} C_VEL
LIN {X 0,Y 89.499,Z 943.087,A -85,B 0,C 180,E1 -27846.116,E2 -27846.116} C_VEL
LIN {X 0,Y 95.721,Z 937.489,A -85,B 0,C 180,E1 -27851.394,E2 -27851.394} C_VEL
LIN {X 0,Y 102.902,Z 930.823,A -85,B 0,C 180,E1 -27855.615,E2 -27855.615} C_VEL
LIN {X 0,Y 104.263,Z 929.734,A -85,B 0,C 180,E1 -27856.163,E2 -27856.163} C_VEL
LIN {X 0,Y 108.716,Z 930.547,A -85,B 0,C 180,E1 -27859.725,E2 -27859.725} C_VEL
LIN {X 0,Y 98.583,Z 921.562,A -85,B 0,C 180,E1 -27866.461,E2 -27866.461} C_VEL
LIN {X 0,Y 95.531,Z 920.923,A -85,B 0,C 180,E1 -27869.004,E2 -27869.004} C_VEL
LIN {X 0,Y 92.71,Z 919.347,A -85,B 0,C 180,E1 -27872.946,E2 -27872.946} C_VEL
LIN {X 0,Y 90.624,Z 917.474,A -85,B 0,C 180,E1 -27877.185,E2 -27877.185} C_VEL
LIN {X 0,Y 88.063,Z 915.273,A -85,B 0,C 180,E1 -27883.363,E2 -27883.363} C_VEL
LIN {X 0,Y 87.821,Z 913.872,A -85,B 0,C 180,E1 -27886.109,E2 -27886.109} C_VEL
LIN {X 0,Y 87.104,Z 911.165,A -85,B 0,C 180,E1 -27893.244,E2 -27893.244} C_VEL
LIN {X 0,Y 86.744,Z 910.582,A -85,B 0,C 180,E1 -27895.856,E2 -27895.856} C_VEL
LIN {X 0,Y 84.597,Z 910.727,A -85,B 0,C 180,E1 -27904.789,E2 -27904.789} C_VEL
LIN {X 0,Y 85.276,Z 909.922,A -85,B 0,C 180,E1 -27907.356,E2 -27907.356} C_VEL
LIN {X 0,Y 88.094,Z 907.349,A -85,B 0,C 180,E1 -27911.485,E2 -27911.485} C_VEL
LIN {X 0,Y 89.878,Z 905.852,A -85,B 0,C 180,E1 -27913.567,E2 -27913.567} C_VEL
LIN {X 0,Y 94.915,Z 902.195,A -85,B 0,C 180,E1 -27919.464,E2 -27919.464} C_VEL
LIN {X 0,Y 98.743,Z 899.402,A -85,B 0,C 180,E1 -27922.229,E2 -27922.229} C_VEL
LIN {X 0,Y 103.555,Z 896.309,A -85,B 0,C 180,E1 -27925.862,E2 -27925.862} C_VEL
LIN {X 0,Y 109.224,Z 892.39,A -85,B 0,C 180,E1 -27928.855,E2 -27928.855} C_VEL
LIN {X 0,Y 116.47,Z 886.858,A -85,B 0,C 180,E1 -27931.643,E2 -27931.643} C_VEL
LIN {X 0,Y 119.374,Z 884.884,A -85,B 0,C 180,E1 -27932.897,E2 -27932.897} C_VEL
LIN {X 0,Y 119.067,Z 885.97,A -85,B 0,C 180,E1 -27933.462,E2 -27933.462} C_VEL
LIN {X 0,Y 113.276,Z 895.172,A -85,B 0,C 180,E1 -27936.205,E2 -27936.205} C_VEL
LIN {X 0,Y 107.106,Z 903.522,A -85,B 0,C 180,E1 -27939.522,E2 -27939.522} C_VEL
LIN {X 0,Y 100.06,Z 911.635,A -85,B 0,C 180,E1 -27943.916,E2 -27943.916} C_VEL
LIN {X 0,Y 93.294,Z 918.483,A -85,B 0,C 180,E1 -27949.218,E2 -27949.218} C_VEL
LIN {X 0,Y 87.135,Z 924.088,A -85,B 0,C 180,E1 -27955.591,E2 -27955.591} C_VEL
LIN {X 0,Y 82.224,Z 927.969,A -85,B 0,C 180,E1 -27961.924,E2 -27961.924} C_VEL
LIN {X 0,Y 78.292,Z 930.832,A -85,B 0,C 180,E1 -27968.922,E2 -27968.922} C_VEL
LIN {X 0,Y 75.171,Z 933.129,A -85,B 0,C 180,E1 -27979.188,E2 -27979.188} C_VEL
LIN {X 0,Y 73.944,Z 933.96,A -85,B 0,C 180,E1 -27989.964,E2 -27989.964} C_VEL
LIN {X 0,Y 75.151,Z 933.185,A -85,B 0,C 180,E1 -28000.743,E2 -28000.743} C_VEL
LIN {X 0,Y 78.244,Z 930.948,A -85,B 0,C 180,E1 -28011.018,E2 -28011.018} C_VEL
LIN {X 0,Y 82.179,Z 928.117,A -85,B 0,C 180,E1 -28018.019,E2 -28018.019} C_VEL
LIN {X 0,Y 87.079,Z 924.282,A -85,B 0,C 180,E1 -28024.36,E2 -28024.36} C_VEL
LIN {X 0,Y 93.19,Z 918.794,A -85,B 0,C 180,E1 -28030.708,E2 -28030.708} C_VEL
LIN {X 0,Y 99.99,Z 911.968,A -85,B 0,C 180,E1 -28036.048,E2 -28036.048} C_VEL
LIN {X 0,Y 107.028,Z 903.925,A -85,B 0,C 180,E1 -28040.45,E2 -28040.45} C_VEL
LIN {X 0,Y 113.184,Z 895.687,A -85,B 0,C 180,E1 -28043.78,E2 -28043.78} C_VEL
LIN {X 0,Y 119.595,Z 885.488,A -85,B 0,C 180,E1 -28046.82,E2 -28046.82} C_VEL
LIN {X 0,Y 124.607,Z 876.054,A -85,B 0,C 180,E1 -28048.893,E2 -28048.893} C_VEL
LIN {X 0,Y 128.404,Z 867.7,A -85,B 0,C 180,E1 -28050.291,E2 -28050.291} C_VEL
LIN {X 0,Y 132.507,Z 856.286,A -85,B 0,C 180,E1 -28051.804,E2 -28051.804} C_VEL
LIN {X 0,Y 135.842,Z 843.256,A -85,B 0,C 180,E1 -28053.158,E2 -28053.158} C_VEL
LIN {X 0,Y 137.855,Z 830.223,A -85,B 0,C 180,E1 -28054.164,E2 -28054.164} C_VEL
LIN {X 0,Y 138.59,Z 821.642,A -85,B 0,C 180,E1 -28054.649,E2 -28054.649} C_VEL
LIN {X 0,Y 135.765,Z 815.023,A -85,B 0,C 180,E1 -28058.383,E2 -28058.383} C_VEL
LIN {X 0,Y 133.185,Z 809.646,A -85,B 0,C 180,E1 -28062.539,E2 -28062.539} C_VEL
LIN {X 0,Y 131.555,Z 806.355,A -85,B 0,C 180,E1 -28065.892,E2 -28065.892} C_VEL
LIN {X 0,Y 130.148,Z 803.241,A -85,B 0,C 180,E1 -28069.892,E2 -28069.892} C_VEL
LIN {X 0,Y 128.905,Z 799.995,A -85,B 0,C 180,E1 -28078.438,E2 -28078.438} C_VEL
LIN {X 0,Y 128.909,Z 800.295,A -85,B 0,C 180,E1 -28080.586,E2 -28080.586} C_VEL
LIN {X 0,Y 129.951,Z 803.199,A -85,B 0,C 180,E1 -28087.575,E2 -28087.575} C_VEL
LIN {X 0,Y 131.545,Z 809.411,A -85,B 0,C 180,E1 -28092.83,E2 -28092.83} C_VEL
LIN {X 0,Y 132.883,Z 814.305,A -85,B 0,C 180,E1 -28095.924,E2 -28095.924} C_VEL
LIN {X 0,Y 134.684,Z 821.081,A -85,B 0,C 180,E1 -28099.331,E2 -28099.331} C_VEL
LIN {X 0,Y 136.246,Z 827.914,A -85,B 0,C 180,E1 -28101.96,E2 -28101.96} C_VEL
LIN {X 0,Y 135.279,Z 848.904,A -85,B 0,C 180,E1 -28103.947,E2 -28103.947} C_VEL
LIN {X 0,Y 134.269,Z 855.785,A -85,B 0,C 180,E1 -28104.47,E2 -28104.47} C_VEL
LIN {X 0,Y 131.323,Z 867.754,A -85,B 0,C 180,E1 -28105.271,E2 -28105.271} C_VEL
LIN {X 0,Y 127.192,Z 879.732,A -85,B 0,C 180,E1 -28106.348,E2 -28106.348} C_VEL
LIN {X 0,Y 122.157,Z 891.173,A -85,B 0,C 180,E1 -28107.857,E2 -28107.857} C_VEL
LIN {X 0,Y 115.549,Z 902.994,A -85,B 0,C 180,E1 -28109.973,E2 -28109.973} C_VEL
LIN {X 0,Y 109.881,Z 911.571,A -85,B 0,C 180,E1 -28112.114,E2 -28112.114} C_VEL
LIN {X 0,Y 103.022,Z 920.485,A -85,B 0,C 180,E1 -28115.104,E2 -28115.104} C_VEL
LIN {X 0,Y 95.389,Z 929.234,A -85,B 0,C 180,E1 -28119.37,E2 -28119.37} C_VEL
LIN {X 0,Y 88.43,Z 936.277,A -85,B 0,C 180,E1 -28124.381,E2 -28124.381} C_VEL
LIN {X 0,Y 82.302,Z 942.146,A -85,B 0,C 180,E1 -28130.51,E2 -28130.51} C_VEL
LIN {X 0,Y 77.569,Z 946.531,A -85,B 0,C 180,E1 -28137.113,E2 -28137.113} C_VEL
LIN {X 0,Y 74.02,Z 950.025,A -85,B 0,C 180,E1 -28144.748,E2 -28144.748} C_VEL
LIN {X 0,Y 72.008,Z 952.556,A -85,B 0,C 180,E1 -28153.014,E2 -28153.014} C_VEL
LIN {X 0,Y 71.593,Z 953.78,A -85,B 0,C 180,E1 -28159.01,E2 -28159.01} C_VEL
LIN {X 0,Y 71.784,Z 954.5,A -85,B 0,C 180,E1 -28164.419,E2 -28164.419} C_VEL
LIN {X 0,Y 72.435,Z 954.844,A -85,B 0,C 180,E1 -28170.037,E2 -28170.037} C_VEL
LIN {X 0,Y 71.831,Z 954.48,A -85,B 0,C 180,E1 -28175.652,E2 -28175.652} C_VEL
LIN {X 0,Y 72.345,Z 952.542,A -85,B 0,C 180,E1 -28186.981,E2 -28186.981} C_VEL
LIN {X 0,Y 74.59,Z 950.014,A -85,B 0,C 180,E1 -28195.125,E2 -28195.125} C_VEL
LIN {X 0,Y 78.474,Z 946.547,A -85,B 0,C 180,E1 -28202.541,E2 -28202.541} C_VEL
LIN {X 0,Y 83.891,Z 942.077,A -85,B 0,C 180,E1 -28208.964,E2 -28208.964} C_VEL
LIN {X 0,Y 90.561,Z 936.483,A -85,B 0,C 180,E1 -28214.339,E2 -28214.339} C_VEL
LIN {X 0,Y 98.376,Z 929.617,A -85,B 0,C 180,E1 -28218.638,E2 -28218.638} C_VEL
LIN {X 0,Y 99.086,Z 928.202,A -85,B 0,C 180,E1 -28219.668,E2 -28219.668} C_VEL
LIN {X 0,Y 87.755,Z 923.964,A -85,B 0,C 180,E1 -28231.281,E2 -28231.281} C_VEL
LIN {X 0,Y 82.292,Z 918.885,A -85,B 0,C 180,E1 -28245.155,E2 -28245.155} C_VEL
LIN {X 0,Y 82.171,Z 914.217,A -85,B 0,C 180,E1 -28257.549,E2 -28257.549} C_VEL
LIN {X 0,Y 82.923,Z 913.005,A -85,B 0,C 180,E1 -28260,E2 -28260} C_VEL
LIN {X 0,Y 85.276,Z 909.922,A -85,B 0,C 180,E1 -28267.356,E2 -28267.356} C_VEL
LIN {X 0,Y 86.933,Z 908.409,A -85,B 0,C 180,E1 -28270.997,E2 -28270.997} C_VEL
LIN {X 0,Y 92.175,Z 905.649,A -85,B 0,C 180,E1 -28281.755,E2 -28281.755} C_VEL
LIN {X 0,Y 95.132,Z 904.075,A -85,B 0,C 180,E1 -28284.686,E2 -28284.686} C_VEL
LIN {X 0,Y 96.317,Z 903.36,A -85,B 0,C 180,E1 -28285.507,E2 -28285.507} C_VEL
LIN {X 0,Y 101.584,Z 900.304,A -85,B 0,C 180,E1 -28288.966,E2 -28288.966} C_VEL
LIN {X 0,Y 107.429,Z 896.669,A -85,B 0,C 180,E1 -28291.698,E2 -28291.698} C_VEL
LIN {X 0,Y 109.286,Z 896.174,A -85,B 0,C 180,E1 -28293.24,E2 -28293.24} C_VEL
LIN {X 0,Y 102.777,Z 904.527,A -85,B 0,C 180,E1 -28296.498,E2 -28296.498} C_VEL
LIN {X 0,Y 95.32,Z 912.64,A -85,B 0,C 180,E1 -28300.872,E2 -28300.872} C_VEL
LIN {X 0,Y 88.092,Z 919.488,A -85,B 0,C 180,E1 -28306.23,E2 -28306.23} C_VEL
LIN {X 0,Y 81.434,Z 925.092,A -85,B 0,C 180,E1 -28312.796,E2 -28312.796} C_VEL
LIN {X 0,Y 76.095,Z 928.972,A -85,B 0,C 180,E1 -28319.433,E2 -28319.433} C_VEL
LIN {X 0,Y 71.779,Z 931.836,A -85,B 0,C 180,E1 -28326.904,E2 -28326.904} C_VEL
LIN {X 0,Y 68.28,Z 934.132,A -85,B 0,C 180,E1 -28338.081,E2 -28338.081} C_VEL
LIN {X 0,Y 66.916,Z 934.962,A -85,B 0,C 180,E1 -28349.96,E2 -28349.96} C_VEL
LIN {X 0,Y 68.259,Z 934.187,A -85,B 0,C 180,E1 -28361.843,E2 -28361.843} C_VEL
LIN {X 0,Y 71.727,Z 931.95,A -85,B 0,C 180,E1 -28373.032,E2 -28373.032} C_VEL
LIN {X 0,Y 76.047,Z 929.119,A -85,B 0,C 180,E1 -28380.507,E2 -28380.507} C_VEL
LIN {X 0,Y 81.374,Z 925.283,A -85,B 0,C 180,E1 -28387.154,E2 -28387.154} C_VEL
LIN {X 0,Y 87.982,Z 919.795,A -85,B 0,C 180,E1 -28393.694,E2 -28393.694} C_VEL
LIN {X 0,Y 95.247,Z 912.969,A -85,B 0,C 180,E1 -28399.094,E2 -28399.094} C_VEL
LIN {X 0,Y 102.696,Z 904.925,A -85,B 0,C 180,E1 -28403.475,E2 -28403.475} C_VEL
LIN {X 0,Y 109.178,Z 896.687,A -85,B 0,C 180,E1 -28406.757,E2 -28406.757} C_VEL
LIN {X 0,Y 115.898,Z 886.486,A -85,B 0,C 180,E1 -28409.729,E2 -28409.729} C_VEL
LIN {X 0,Y 121.125,Z 877.052,A -85,B 0,C 180,E1 -28411.741,E2 -28411.741} C_VEL
LIN {X 0,Y 125.712,Z 866.993,A -85,B 0,C 180,E1 -28413.387,E2 -28413.387} C_VEL
LIN {X 0,Y 130.214,Z 854.531,A -85,B 0,C 180,E1 -28414.846,E2 -28414.846} C_VEL
LIN {X 0,Y 133.225,Z 842.248,A -85,B 0,C 180,E1 -28416.041,E2 -28416.041} C_VEL
LIN {X 0,Y 135.152,Z 829.242,A -85,B 0,C 180,E1 -28416.954,E2 -28416.954} C_VEL
LIN {X 0,Y 135.509,Z 825.322,A -85,B 0,C 180,E1 -28417.187,E2 -28417.187} C_VEL
LIN {X 0,Y 132.994,Z 819.102,A -85,B 0,C 180,E1 -28421.114,E2 -28421.114} C_VEL
LIN {X 0,Y 131.162,Z 815.117,A -85,B 0,C 180,E1 -28424.621,E2 -28424.621} C_VEL
LIN {X 0,Y 130.117,Z 812.819,A -85,B 0,C 180,E1 -28427.126,E2 -28427.126} C_VEL
LIN {X 0,Y 128.964,Z 810.023,A -85,B 0,C 180,E1 -28430.887,E2 -28430.887} C_VEL
LIN {X 0,Y 128.026,Z 807.157,A -85,B 0,C 180,E1 -28438.427,E2 -28438.427} C_VEL
LIN {X 0,Y 128.027,Z 807.48,A -85,B 0,C 180,E1 -28440.59,E2 -28440.59} C_VEL
LIN {X 0,Y 128.798,Z 809.879,A -85,B 0,C 180,E1 -28446.56,E2 -28446.56} C_VEL
LIN {X 0,Y 130.077,Z 815.794,A -85,B 0,C 180,E1 -28451.591,E2 -28451.591} C_VEL
LIN {X 0,Y 131.165,Z 820.522,A -85,B 0,C 180,E1 -28454.546,E2 -28454.546} C_VEL
LIN {X 0,Y 132.711,Z 827.301,A -85,B 0,C 180,E1 -28457.933,E2 -28457.933} C_VEL
LIN {X 0,Y 133.464,Z 831.163,A -85,B 0,C 180,E1 -28459.446,E2 -28459.446} C_VEL
LIN {X 0,Y 132.244,Z 849.806,A -85,B 0,C 180,E1 -28461.229,E2 -28461.229} C_VEL
LIN {X 0,Y 131.15,Z 856.337,A -85,B 0,C 180,E1 -28461.722,E2 -28461.722} C_VEL
LIN {X 0,Y 127.608,Z 869.467,A -85,B 0,C 180,E1 -28462.604,E2 -28462.604} C_VEL
LIN {X 0,Y 122.829,Z 882.009,A -85,B 0,C 180,E1 -28463.788,E2 -28463.788} C_VEL
LIN {X 0,Y 117.484,Z 893.038,A -85,B 0,C 180,E1 -28465.267,E2 -28465.267} C_VEL
LIN {X 0,Y 110.671,Z 904.297,A -85,B 0,C 180,E1 -28467.307,E2 -28467.307} C_VEL
LIN {X 0,Y 104.819,Z 912.521,A -85,B 0,C 180,E1 -28469.41,E2 -28469.41} C_VEL
LIN {X 0,Y 96.338,Z 922.583,A -85,B 0,C 180,E1 -28473.028,E2 -28473.028} C_VEL
LIN {X 0,Y 88.46,Z 930.739,A -85,B 0,C 180,E1 -28477.449,E2 -28477.449} C_VEL
LIN {X 0,Y 81.307,Z 937.326,A -85,B 0,C 180,E1 -28482.769,E2 -28482.769} C_VEL
LIN {X 0,Y 75.162,Z 942.629,A -85,B 0,C 180,E1 -28489.166,E2 -28489.166} C_VEL
LIN {X 0,Y 70.143,Z 946.806,A -85,B 0,C 180,E1 -28496.607,E2 -28496.607} C_VEL
LIN {X 0,Y 66.602,Z 949.973,A -85,B 0,C 180,E1 -28505.08,E2 -28505.08} C_VEL
LIN {X 0,Y 64.568,Z 952.705,A -85,B 0,C 180,E1 -28517.47,E2 -28517.47} C_VEL
LIN {X 0,Y 64.698,Z 953.484,A -85,B 0,C 180,E1 -28523.806,E2 -28523.806} C_VEL
LIN {X 0,Y 65.332,Z 953.83,A -85,B 0,C 180,E1 -28530.041,E2 -28530.041} C_VEL
LIN {X 0,Y 64.759,Z 953.466,A -85,B 0,C 180,E1 -28536.271,E2 -28536.271} C_VEL
LIN {X 0,Y 65.539,Z 951.521,A -85,B 0,C 180,E1 -28548.808,E2 -28548.808} C_VEL
LIN {X 0,Y 68.22,Z 948.999,A -85,B 0,C 180,E1 -28557.661,E2 -28557.661} C_VEL
LIN {X 0,Y 72.591,Z 945.534,A -85,B 0,C 180,E1 -28565.556,E2 -28565.556} C_VEL
LIN {X 0,Y 78.522,Z 941.068,A -85,B 0,C 180,E1 -28572.208,E2 -28572.208} C_VEL
LIN {X 0,Y 85.67,Z 935.478,A -85,B 0,C 180,E1 -28577.63,E2 -28577.63} C_VEL
LIN {X 0,Y 89.792,Z 932.113,A -85,B 0,C 180,E1 -28579.949,E2 -28579.949} C_VEL
LIN {X 0,Y 89.981,Z 930.872,A -85,B 0,C 180,E1 -28581.329,E2 -28581.329} C_VEL
LIN {X 0,Y 82.699,Z 928.241,A -85,B 0,C 180,E1 -28589.343,E2 -28589.343} C_VEL
LIN {X 0,Y 76.718,Z 923.389,A -85,B 0,C 180,E1 -28604.049,E2 -28604.049} C_VEL
LIN {X 0,Y 76.119,Z 919.838,A -85,B 0,C 180,E1 -28614.703,E2 -28614.703} C_VEL
LIN {X 0,Y 80.78,Z 913.857,A -85,B 0,C 180,E1 -28630.021,E2 -28630.021} C_VEL
LIN {X 0,Y 86.102,Z 909.842,A -85,B 0,C 180,E1 -28636.6,E2 -28636.6} C_VEL
LIN {X 0,Y 91.822,Z 906.219,A -85,B 0,C 180,E1 -28642.501,E2 -28642.501} C_VEL
LIN {X 0,Y 96.317,Z 903.36,A -85,B 0,C 180,E1 -28645.507,E2 -28645.507} C_VEL
LIN {X 0,Y 97.364,Z 903.013,A -85,B 0,C 180,E1 -28646.744,E2 -28646.744} C_VEL
LIN {X 0,Y 97.648,Z 903.77,A -85,B 0,C 180,E1 -28648.659,E2 -28648.659} C_VEL
LIN {X 0,Y 96.786,Z 905.902,A -85,B 0,C 180,E1 -28651.108,E2 -28651.108} C_VEL
LIN {X 0,Y 95.442,Z 907.958,A -85,B 0,C 180,E1 -28652.903,E2 -28652.903} C_VEL
LIN {X 0,Y 93.3,Z 910.673,A -85,B 0,C 180,E1 -28654.962,E2 -28654.962} C_VEL
LIN {X 0,Y 88.387,Z 915.932,A -85,B 0,C 180,E1 -28658.998,E2 -28658.998} C_VEL
LIN {X 0,Y 85.667,Z 918.407,A -85,B 0,C 180,E1 -28661.007,E2 -28661.007} C_VEL
LIN {X 0,Y 78.064,Z 924.539,A -85,B 0,C 180,E1 -28667.487,E2 -28667.487} C_VEL
LIN {X 0,Y 74.009,Z 927.47,A -85,B 0,C 180,E1 -28671.842,E2 -28671.842} C_VEL
LIN {X 0,Y 68.397,Z 931.02,A -85,B 0,C 180,E1 -28679.042,E2 -28679.042} C_VEL
LIN {X 0,Y 65.372,Z 932.839,A -85,B 0,C 180,E1 -28684.487,E2 -28684.487} C_VEL
LIN {X 0,Y 61.421,Z 935.135,A -85,B 0,C 180,E1 -28696.727,E2 -28696.727} C_VEL
LIN {X 0,Y 59.888,Z 935.965,A -85,B 0,C 180,E1 -28709.955,E2 -28709.955} C_VEL
LIN {X 0,Y 61.397,Z 935.19,A -85,B 0,C 180,E1 -28723.189,E2 -28723.189} C_VEL
LIN {X 0,Y 65.317,Z 932.952,A -85,B 0,C 180,E1 -28735.445,E2 -28735.445} C_VEL
LIN {X 0,Y 70.083,Z 930.121,A -85,B 0,C 180,E1 -28743.425,E2 -28743.425} C_VEL
LIN {X 0,Y 75.891,Z 926.285,A -85,B 0,C 180,E1 -28750.36,E2 -28750.36} C_VEL
LIN {X 0,Y 83.042,Z 920.796,A -85,B 0,C 180,E1 -28757.046,E2 -28757.046} C_VEL
LIN {X 0,Y 90.8,Z 913.97,A -85,B 0,C 180,E1 -28762.447,E2 -28762.447} C_VEL
LIN {X 0,Y 98.675,Z 905.926,A -85,B 0,C 180,E1 -28766.756,E2 -28766.756} C_VEL
LIN {X 0,Y 105.489,Z 897.686,A -85,B 0,C 180,E1 -28769.951,E2 -28769.951} C_VEL
LIN {X 0,Y 112.519,Z 887.485,A -85,B 0,C 180,E1 -28772.821,E2 -28772.821} C_VEL
LIN {X 0,Y 117.961,Z 878.05,A -85,B 0,C 180,E1 -28774.748,E2 -28774.748} C_VEL
LIN {X 0,Y 122.725,Z 867.99,A -85,B 0,C 180,E1 -28776.322,E2 -28776.322} C_VEL
LIN {X 0,Y 127.162,Z 856.234,A -85,B 0,C 180,E1 -28777.621,E2 -28777.621} C_VEL
LIN {X 0,Y 130.429,Z 843.758,A -85,B 0,C 180,E1 -28778.821,E2 -28778.821} C_VEL
LIN {X 0,Y 132.464,Z 830.97,A -85,B 0,C 180,E1 -28779.724,E2 -28779.724} C_VEL
LIN {X 0,Y 132.598,Z 828.951,A -85,B 0,C 180,E1 -28779.947,E2 -28779.947} C_VEL
LIN {X 0,Y 130.626,Z 823.763,A -85,B 0,C 180,E1 -28783.693,E2 -28783.693} C_VEL
LIN {X 0,Y 129.019,Z 819.762,A -85,B 0,C 180,E1 -28787.614,E2 -28787.614} C_VEL
LIN {X 0,Y 127.88,Z 816.86,A -85,B 0,C 180,E1 -28791.664,E2 -28791.664} C_VEL
LIN {X 0,Y 127.148,Z 814.311,A -85,B 0,C 180,E1 -28798.416,E2 -28798.416} C_VEL
LIN {X 0,Y 127.157,Z 814.733,A -85,B 0,C 180,E1 -28800.891,E2 -28800.891} C_VEL
LIN {X 0,Y 127.699,Z 816.672,A -85,B 0,C 180,E1 -28805.626,E2 -28805.626} C_VEL
LIN {X 0,Y 128.622,Z 821.942,A -85,B 0,C 180,E1 -28810.148,E2 -28810.148} C_VEL
LIN {X 0,Y 129.739,Z 827.686,A -85,B 0,C 180,E1 -28813.709,E2 -28813.709} C_VEL
LIN {X 0,Y 130.82,Z 833.759,A -85,B 0,C 180,E1 -28816.538,E2 -28816.538} C_VEL
LIN {X 0,Y 130.934,Z 834.415,A -85,B 0,C 180,E1 -28816.81,E2 -28816.81} C_VEL
LIN {X 0,Y 129.648,Z 849.765,A -85,B 0,C 180,E1 -28818.309,E2 -28818.309} C_VEL
LIN {X 0,Y 128.446,Z 856.433,A -85,B 0,C 180,E1 -28818.827,E2 -28818.827} C_VEL
LIN {X 0,Y 124.758,Z 869.281,A -85,B 0,C 180,E1 -28819.655,E2 -28819.655} C_VEL
LIN {X 0,Y 120.12,Z 880.993,A -85,B 0,C 180,E1 -28820.662,E2 -28820.662} C_VEL
LIN {X 0,Y 114.622,Z 892.026,A -85,B 0,C 180,E1 -28822.041,E2 -28822.041} C_VEL
LIN {X 0,Y 107.59,Z 903.284,A -85,B 0,C 180,E1 -28823.934,E2 -28823.934} C_VEL
LIN {X 0,Y 101.521,Z 911.512,A -85,B 0,C 180,E1 -28825.917,E2 -28825.917} C_VEL
LIN {X 0,Y 92.654,Z 921.571,A -85,B 0,C 180,E1 -28829.339,E2 -28829.339} C_VEL
LIN {X 0,Y 84.322,Z 929.726,A -85,B 0,C 180,E1 -28833.606,E2 -28833.606} C_VEL
LIN {X 0,Y 76.632,Z 936.308,A -85,B 0,C 180,E1 -28838.842,E2 -28838.842} C_VEL
LIN {X 0,Y 69.896,Z 941.608,A -85,B 0,C 180,E1 -28845.321,E2 -28845.321} C_VEL
LIN {X 0,Y 64.297,Z 945.788,A -85,B 0,C 180,E1 -28853.1,E2 -28853.1} C_VEL
LIN {X 0,Y 60.166,Z 948.949,A -85,B 0,C 180,E1 -28862.197,E2 -28862.197} C_VEL
LIN {X 0,Y 57.585,Z 951.681,A -85,B 0,C 180,E1 -28875.921,E2 -28875.921} C_VEL
LIN {X 0,Y 57.598,Z 952.464,A -85,B 0,C 180,E1 -28883.039,E2 -28883.039} C_VEL
LIN {X 0,Y 58.23,Z 952.817,A -85,B 0,C 180,E1 -28890.046,E2 -28890.046} C_VEL
LIN {X 0,Y 57.697,Z 952.451,A -85,B 0,C 180,E1 -28897.043,E2 -28897.043} C_VEL
LIN {X 0,Y 58.838,Z 950.504,A -85,B 0,C 180,E1 -28911.045,E2 -28911.045} C_VEL
LIN {X 0,Y 62.014,Z 947.984,A -85,B 0,C 180,E1 -28920.71,E2 -28920.71} C_VEL
LIN {X 0,Y 66.946,Z 944.521,A -85,B 0,C 180,E1 -28929.09,E2 -28929.09} C_VEL
LIN {X 0,Y 73.445,Z 940.059,A -85,B 0,C 180,E1 -28935.912,E2 -28935.912} C_VEL
LIN {X 0,Y 81.086,Z 934.47,A -85,B 0,C 180,E1 -28941.313,E2 -28941.313} C_VEL
LIN {X 0,Y 81.19,Z 933.51,A -85,B 0,C 180,E1 -28942.704,E2 -28942.704} C_VEL
LIN {X 0,Y 74.748,Z 930.63,A -85,B 0,C 180,E1 -28951.958,E2 -28951.958} C_VEL
LIN {X 0,Y 70.235,Z 925.813,A -85,B 0,C 180,E1 -28968.456,E2 -28968.456} C_VEL
LIN {X 0,Y 71.082,Z 922.254,A -85,B 0,C 180,E1 -28980,E2 -28980} C_VEL
LIN {X 0,Y 76.454,Z 917.388,A -85,B 0,C 180,E1 -28993.286,E2 -28993.286} C_VEL
LIN {X 0,Y 82.366,Z 913.561,A -85,B 0,C 180,E1 -28999.957,E2 -28999.957} C_VEL
LIN {X 0,Y 88.828,Z 909.977,A -85,B 0,C 180,E1 -29005.796,E2 -29005.796} C_VEL
LIN {X 0,Y 96.702,Z 905.67,A -85,B 0,C 180,E1 -29010.58,E2 -29010.58} C_VEL
LIN {X 0,Y 100.136,Z 903.954,A -85,B 0,C 180,E1 -29012.582,E2 -29012.582} C_VEL
LIN {X 0,Y 92.163,Z 912.439,A -85,B 0,C 180,E1 -29016.761,E2 -29016.761} C_VEL
LIN {X 0,Y 85.667,Z 918.407,A -85,B 0,C 180,E1 -29021.007,E2 -29021.007} C_VEL
LIN {X 0,Y 81.809,Z 921.428,A -85,B 0,C 180,E1 -29023.283,E2 -29023.283} C_VEL
LIN {X 0,Y 74.297,Z 925.97,A -85,B 0,C 180,E1 -29026.704,E2 -29026.704} C_VEL
LIN {X 0,Y 66.786,Z 929.784,A -85,B 0,C 180,E1 -29031.019,E2 -29031.019} C_VEL
LIN {X 0,Y 63.119,Z 931.664,A -85,B 0,C 180,E1 -29034.789,E2 -29034.789} C_VEL
LIN {X 0,Y 59.107,Z 933.842,A -85,B 0,C 180,E1 -29041.551,E2 -29041.551} C_VEL
LIN {X 0,Y 54.604,Z 936.138,A -85,B 0,C 180,E1 -29055.034,E2 -29055.034} C_VEL
LIN {X 0,Y 52.86,Z 936.968,A -85,B 0,C 180,E1 -29069.949,E2 -29069.949} C_VEL
LIN {X 0,Y 54.578,Z 936.192,A -85,B 0,C 180,E1 -29084.872,E2 -29084.872} C_VEL
LIN {X 0,Y 59.047,Z 933.954,A -85,B 0,C 180,E1 -29098.377,E2 -29098.377} C_VEL
LIN {X 0,Y 64.334,Z 931.122,A -85,B 0,C 180,E1 -29106.875,E2 -29106.875} C_VEL
LIN {X 0,Y 70.682,Z 927.286,A -85,B 0,C 180,E1 -29114.052,E2 -29114.052} C_VEL
LIN {X 0,Y 78.422,Z 921.797,A -85,B 0,C 180,E1 -29120.807,E2 -29120.807} C_VEL
LIN {X 0,Y 86.696,Z 914.97,A -85,B 0,C 180,E1 -29126.132,E2 -29126.132} C_VEL
LIN {X 0,Y 95.004,Z 906.926,A -85,B 0,C 180,E1 -29130.303,E2 -29130.303} C_VEL
LIN {X 0,Y 102.151,Z 898.686,A -85,B 0,C 180,E1 -29133.365,E2 -29133.365} C_VEL
LIN {X 0,Y 109.487,Z 888.484,A -85,B 0,C 180,E1 -29136.095,E2 -29136.095} C_VEL
LIN {X 0,Y 115.723,Z 877.986,A -85,B 0,C 180,E1 -29138.072,E2 -29138.072} C_VEL
LIN {X 0,Y 120.514,Z 867.991,A -85,B 0,C 180,E1 -29139.518,E2 -29139.518} C_VEL
LIN {X 0,Y 125.137,Z 855.779,A -85,B 0,C 180,E1 -29140.76,E2 -29140.76} C_VEL
LIN {X 0,Y 128.297,Z 843.582,A -85,B 0,C 180,E1 -29141.835,E2 -29141.835} C_VEL
LIN {X 0,Y 130.049,Z 833.078,A -85,B 0,C 180,E1 -29142.589,E2 -29142.589} C_VEL
LIN {X 0,Y 128.515,Z 828.574,A -85,B 0,C 180,E1 -29146.359,E2 -29146.359} C_VEL
LIN {X 0,Y 127.55,Z 825.948,A -85,B 0,C 180,E1 -29149.283,E2 -29149.283} C_VEL
LIN {X 0,Y 126.825,Z 823.691,A -85,B 0,C 180,E1 -29152.436,E2 -29152.436} C_VEL
LIN {X 0,Y 126.273,Z 821.438,A -85,B 0,C 180,E1 -29158.405,E2 -29158.405} C_VEL
LIN {X 0,Y 126.279,Z 821.879,A -85,B 0,C 180,E1 -29160.897,E2 -29160.897} C_VEL
LIN {X 0,Y 126.635,Z 823.454,A -85,B 0,C 180,E1 -29164.675,E2 -29164.675} C_VEL
LIN {X 0,Y 127.283,Z 828.324,A -85,B 0,C 180,E1 -29168.834,E2 -29168.834} C_VEL
LIN {X 0,Y 128.16,Z 834.215,A -85,B 0,C 180,E1 -29172.369,E2 -29172.369} C_VEL
LIN {X 0,Y 128.665,Z 837.647,A -85,B 0,C 180,E1 -29174.029,E2 -29174.029} C_VEL
LIN {X 0,Y 127.176,Z 851.007,A -85,B 0,C 180,E1 -29175.388,E2 -29175.388} C_VEL
